// TIA Portal project "BancoProvaProfilometroSpessimetro_V15" (V15)

(* hardware
DEVICE "S71500/ET200MP station_1"  S7-1500 station
   slot 0: "Telaio di montaggio_0"  Rack  6ES7 590-1***0-0AA0
   slot 1: "PLC_1"  CPU 1515-2 PN  6ES7 515-2AM01-0AB0  V2.1
      slot 3: "Display CPU_1"  6ES7591-1BA00-0AA0
DEVICE "GSD device_1"  GSD.Device.PN
   slot 0: "Telaio di montaggio"  Rail  V1.0
   slot 0: "IAI-PRT"  IAI-PRT
   slot 1: "Input 1 word_1"  IAI-PRT
   slot 2: "Input 1 word_2"  IAI-PRT
   slot 3: "Input 1 word_3"  IAI-PRT
   slot 4: "Input 1 word_4"  IAI-PRT
   slot 5: "Input 1 word_5"  IAI-PRT
   slot 6: "Input 1 word_6"  IAI-PRT
   slot 7: "Input 1 word_7"  IAI-PRT
   slot 8: "Input 1 word_8"  IAI-PRT
   slot 9: "Input 1 word_9"  IAI-PRT
   slot 10: "Input 1 word_10"  IAI-PRT
   slot 11: "Input 1 word_11"  IAI-PRT
   slot 12: "Input 1 word_12"  IAI-PRT
   slot 13: "Input 1 word_13"  IAI-PRT
   slot 14: "Input 1 word_14"  IAI-PRT
   slot 15: "Input 1 word_15"  IAI-PRT
   slot 16: "Input 1 word_16"  IAI-PRT
   slot 17: "Output 1 word_1"  IAI-PRT
   slot 18: "Output 1 word_2"  IAI-PRT
   slot 19: "Output 1 word_3"  IAI-PRT
   slot 20: "Output 1 word_4"  IAI-PRT
   slot 21: "Output 1 word_5"  IAI-PRT
   slot 22: "Output 1 word_6"  IAI-PRT
   slot 23: "Output 1 word_7"  IAI-PRT
   slot 24: "Output 1 word_8"  IAI-PRT
   slot 25: "Output 1 word_9"  IAI-PRT
   slot 26: "Output 1 word_10"  IAI-PRT
   slot 27: "Output 1 word_11"  IAI-PRT
   slot 28: "Output 1 word_12"  IAI-PRT
   slot 29: "Output 1 word_13"  IAI-PRT
   slot 30: "Output 1 word_14"  IAI-PRT
   slot 31: "Output 1 word_15"  IAI-PRT
   slot 32: "Output 1 word_16"  IAI-PRT
DEVICE "HMI_1"  KTP400 Comfort
   slot 0: "HMI_1"  KTP400 Comfort  6AV2 124-2DC01-0AX0  15.0.0.0
   slot 1: "HMI_RT_1"  KTP400 Comfort  6AV2 124-2DC01-0AX0  15.0.0.0
   slot 5: "HMI_1.IE_CP_1"  PROFINET Interface  15.0.0.0
      slot 1: "PROFINET Interface_1"  PROFINET Interface
         slot 1: "Porta_1"  Port
   slot 7: "HMI_1.MPI/DP_CP_1"  MPI/DP Interface  15.0.0.0
DEVICE "GSD device_2"  GSD.Device.PN
   slot 0: "Telaio di montaggio"  Rail  V1.0
   slot 0: "dl-pn1"  DL-PN1  1.00
*)

// ===== PLC "PLC_1"  CPU 1515-2 PN =====

VAR_GLOBAL   // PLC tag table "IO_IAI_Controller"
   "RMDS" AT %I30.0 : Bool;   // Stato del segnale operativo - 0: Auto - 1: Manu
   "TRQS" AT %I30.1 : Bool;   // Stato del livello di coppia - questo segnale diventerà vero quando il motore raggiungerà il livello di soglia
   "LOAD" AT %I30.2 : Bool;   // Questo segnale diventerà vero quando la coppia di comando supera la soglia, mentre l'attuatore si trova al interno del range di verifica
   "PZONE" AT %I30.3 : Bool;   // Questo segnale diventerà vero quando dopo l'immissione di un comando di position movement , la posizione effettiva sarà nel range specificato. Uscito da tale range il segnale diventerà falso
   "ZONE1" AT %I30.4 : Bool;   // Questo segnale diventerà vero una volta entrati nel range specificato e sempre solo dopo che l'asse si sia mosso dalla zona 0 (Home) fino alla zona desiderata. Uscito da tale range il contatto diventa falso
   "ZONE2" AT %I30.5 : Bool;   // Questo segnale diventerà vero una volta entrati nel range specificato e sempre solo dopo che l'asse si sia mosso dalla zona 0 (Home) fino alla zona desiderata. Uscito da tale range il contatto diventa falso
   "PWRT" AT %I30.6 : Bool;   // Scrittura della posizione corrente - Se il segnale rimane vero per più di 20ms la posizione attuale verrà salvata da pc1 a pc32
   "EMGS" AT %I30.7 : Bool;   // Stop di emergenza, se viene premuto questa entrata diventa vera
   "PEND" AT %I31.0 : Bool;   // Diventa vero quando il posizionamento è stato terminato
   "HEND" AT %I31.1 : Bool;   // Diventa vero quando viene premuto HOME e l'attuatore è effettivamente nella posizione HOME
   "MOVE" AT %I31.2 : Bool;   // Determina il movimento generico del asse
   "ALM" AT %I31.3 : Bool;   // Contatto NC - se è presente un evento di allarme il segnale diventa falso, in condizioni normali è vero
   "SV" AT %I31.4 : Bool;   // Se vero, indica che il controller è pronto
   "PSFL" AT %I31.5 : Bool;   // -
   "PUSH" AT %I31.6 : Bool;   // -
   "GHMS" AT %I31.7 : Bool;   // -
   "COMMAND_CURRENT" AT %ID4 : DWord;   // Comando attuale
   "CURRENT_SPEED" AT %ID8 : DWord;   // Velocità attuale
   "CSTR" AT %Q31.0 : Bool;   // Start del comando
   "HOME" AT %Q31.1 : Bool;   // L'operazione di ritorno viene avviata a un fronte di salita di questo segnale
   "STP" AT %Q31.2 : Bool;   // ON: l'attuatore può essere spostato, OFF: l'attuatore decelera fino all'arresto
   "RES" AT %Q31.3 : Bool;   // Un allarme viene resettato su un fronte di salita di questo segnale
   "SON" AT %Q31.4 : Bool;   // Servo ON - abilita il servo motore
   "JISL" AT %Q31.5 : Bool;   // Abilita le operazioni manuali (Controller su MANUAL)
   "JVEL" AT %Q31.6 : Bool;
   "JOGneg" AT %Q31.7 : Bool;   // Muovo in libertà l'asse, verso negativo
   "JOGpos" AT %Q30.0 : Bool;   // Muovo in libertà l'asse, verso positivo
   "RMDO" AT %Q30.6 : Bool;   // Questo segnale cambia la modalità operativa tra AUTO e MANU
   "BKRL" AT %Q30.7 : Bool;   // Questo segnale viene utilizzato su un attuatore dotato di un freno per forzarne il rilascio
   "TARGET_POSITION" AT %QD0 : DInt;   // Posizione desiderata
   "POSITION_BAND" AT %QD4 : DInt;   // Banda di posizione desiderata
   "SPEED" AT %QD8 : DInt;   // Veocità simulata
   "ZONE_OUTPUT_POS_positive" AT %QD12 : DInt;
   "ZONE_OUTPUT_POS_negative" AT %QD16 : DInt;
   "PRESSING_CURRENT_LIMIT" AT %QD32 : DInt;
   "LOAD_CURRENT_THRESHOLD" AT %QD36 : DInt;
   "Tag_7" AT %QD26 : DWord;
   "Tag_8" AT %QW24 : Word;
   "ACELERATION" AT %QW20 : Int;   // Accelerzione simulata
   "DECELERATION" AT %QW22 : Int;   // Decelerazione simulata
   "M_SON_AXIS" AT %M100.0 : Bool;
   "M_STR_AXIS" AT %M100.1 : Bool;
   "M_DSTR_ON" AT %M100.2 : Bool;
   "Tag_4" AT %MW32 : Word;
   "Tag_6" AT %MW202 : Word;
   "Tag_12" AT %M204.3 : Bool;
   "Tag_13" AT %MW206 : Word;
   "M_REQUEST_STATUS" AT %M300.0 : Bool;
   "M_RETURN_HOME" AT %M400.0 : Bool;
   "M_JOG_POS" AT %M100.3 : Bool;
   "M_JOG_NEG" AT %M100.4 : Bool;
   "M_RESET_ALLARM" AT %M100.5 : Bool;
   "ON" AT %M106.0 : Bool;
   "Clock_Byte" AT %MB0 : Byte;
   "Clock_10Hz" AT %M0.0 : Bool;
   "Clock_5Hz" AT %M0.1 : Bool;
   "Clock_2.5Hz" AT %M0.2 : Bool;
   "Clock_2Hz" AT %M0.3 : Bool;
   "Clock_1.25Hz" AT %M0.4 : Bool;
   "Clock_1Hz" AT %M0.5 : Bool;
   "Clock_0.625Hz" AT %M0.6 : Bool;
   "Clock_0.5Hz" AT %M0.7 : Bool;
   "Tag_1" AT %M120.0 : Bool;
   "System_Byte" AT %MB1 : Byte;
   "FirstScan" AT %M1.0 : Bool;
   "DiagStatusUpdate" AT %M1.1 : Bool;
   "AlwaysTRUE" AT %M1.2 : Bool;
   "AlwaysFALSE" AT %M1.3 : Bool;
   "ReportFF" AT %M410.0 : Bool;
   "SelectOPMode" AT %M10.0 : Bool;   // Seleziono il modo operativo
   "OPMode_Set" AT %M10.1 : Bool;   // Porto a 1 il modo operativo
   "OPMode_Reset" AT %M10.2 : Bool;   // Porto a 0 il modo operativo
   "OPMode_ResetCTU" AT %M10.3 : Bool;   // Resetto il conteggio di Counter_JogAuto
   "Rnd_Seed" AT %MW100 : Word;
   "Rnd_Restart" AT %M20.0 : Bool;
   "Rnd_Record" AT %MW101 : Word;
   "Rnd_Seed_Pos" AT %MW102 : Word;
   "Rnd_Record_Pos" AT %MW113 : Word;
   "Restart_Sim" AT %M30.0 : Bool;
   "Restart_Sim_Set" AT %M30.1 : Bool;
   "Restart_Sim_Reset" AT %M30.2 : Bool;
   "Restart_Sim_RCTU" AT %M30.3 : Bool;
   "PreviusPosition" AT %MD103 : DWord;
   "ChangeDetected" AT %M40.0 : Bool;
   "Tag_5" AT %MD104 : DWord;
   "ResetSQLChangeValue" AT %M50.0 : Bool;
   "REQ_IL1000_Set" AT %M60.0 : Bool;
   "REQ_IL1000_Reset" AT %M60.1 : Bool;
   "REQ_IL1000_ResCTU" AT %M60.2 : Bool;
   "Tag_2" AT %M70.0 : Bool;
   "Tag_3" AT %M80.0 : Bool;
   "Tag_9" AT %MD45 : DWord;
   "Tag_10" AT %MD46 : DWord;
   "Tag_11" AT %M5.0 : Bool;
   "Simu_Timer" AT %M6.0 : Bool;
   "RawPosition" AT %ID0 : DWord;
   "M_SON" AT %M101.0 : Bool;   // Merker - Start Servo
   "Cock_10Hz_Neg" AT %M321.0 : Bool;
   "Tag_16" AT %M102.0 : Bool;
END_VAR

VAR_GLOBAL   // PLC tag table "Keyence"
   "SensorIN" AT %IW32 : Word;
   "ERROR_IL1000" AT %M204.2 : Bool;
   "RECORD_IL1000" AT %MD215 : DInt;
   "LEN_IL1000" AT %MD210 : DWord;
   "STATUS_IL1000" AT %MD206 : DWord;
   "VALID_IL1000" AT %M204.0 : Bool;
   "BUSY_IL1000" AT %M204.1 : Bool;
   "REQ_IL1000" AT %M500.0 : Bool;
   "IL_100_ST" AT %M100.6 : Bool;
END_VAR

// folder: Database/Istanze

DATA_BLOCK "Output_DB"   // DB7
{ S7_Optimized_Access := 'TRUE' }
AUTHOR : Valentino-Fabbri
VERSION : 0.1
// stored: InstanceOfName Output
"Output"
BEGIN
END_DATA_BLOCK

DATA_BLOCK "Jog Manager_DB"   // DB8
{ S7_Optimized_Access := 'TRUE' }
AUTHOR : Valentino-Fabbri
VERSION : 0.1
// stored: InstanceOfName Jog Manager
"Jog Manager"
BEGIN
END_DATA_BLOCK

DATA_BLOCK "Position Move_DB"   // DB9
{ S7_Optimized_Access := 'TRUE' }
AUTHOR : Valentino-Fabbri
VERSION : 0.1
// stored: InstanceOfName Position Move
"Position Move"
BEGIN
END_DATA_BLOCK

DATA_BLOCK "Speed Move_DB"   // DB10
{ S7_Optimized_Access := 'TRUE' }
AUTHOR : Valentino-Fabbri
VERSION : 0.1
// stored: InstanceOfName Speed Move
"Speed Move"
BEGIN
END_DATA_BLOCK

DATA_BLOCK "DoubleTapButton2_DB_3"   // DB12
{ S7_Optimized_Access := 'TRUE' }
VERSION : 0.1
// stored: InstanceOfName DoubleTapButton2
"DoubleTapButton2"
BEGIN
END_DATA_BLOCK

DATA_BLOCK "DoubleTapButton2_DB"   // DB21
{ S7_Optimized_Access := 'TRUE' }
VERSION : 0.1
// stored: InstanceOfName DoubleTapButton2
"DoubleTapButton2"
BEGIN
END_DATA_BLOCK

DATA_BLOCK "DoubleTapButton2_DB_1"   // DB22
{ S7_Optimized_Access := 'TRUE' }
VERSION : 0.1
// stored: InstanceOfName DoubleTapButton2
"DoubleTapButton2"
BEGIN
END_DATA_BLOCK

DATA_BLOCK "DoubleTapButton2_DB_2"   // DB23
{ S7_Optimized_Access := 'TRUE' }
VERSION : 0.1
// stored: InstanceOfName DoubleTapButton2
"DoubleTapButton2"
BEGIN
END_DATA_BLOCK

DATA_BLOCK "CollisionMovement_DB"   // DB24
{ S7_Optimized_Access := 'TRUE' }
AUTHOR : Valentino-Fabbri
VERSION : 0.1
// stored: InstanceOfName CollisionMovement
"CollisionMovement"
BEGIN
END_DATA_BLOCK

DATA_BLOCK "Input_DB"   // DB26
{ S7_Optimized_Access := 'TRUE' }
AUTHOR : Valentino-Fabbri
VERSION : 0.1
// stored: InstanceOfName Input
"Input"
BEGIN
END_DATA_BLOCK

// folder: Database/Static

DATA_BLOCK "IAI_DATI"   // DB2
{ S7_Optimized_Access := 'TRUE' }
VERSION : 0.1
   VAR
      "TargetPosition 1" : DInt := 0;   // Posizione desiderata - impostata a metà
      "TargetPosition 2" : Real := 0.0;
      "TargetPosition 2 Out" : DInt;
      PositionBand : Real := 10000.0;   // Margine di errore sulla posizione desiderata
      PositionBandOut : DInt;
      Speed : Real := 3000.0;   // Velocità espressa in mm/s
      SpeedOut : DInt := 0;
      Aceleration : Real := 1.0;   // Accellerazione
      AcelerationOut : DInt := 0;
      Deceleration : Real := 1.0;   // Decellerazione
      DecelerationOut : DInt := 0;
      ZonePos : Real := 10000.0;
      ZonePosOut : DInt := 0;
      ZoneNeg : Real := 10000.0;
      ZoneNegOut : DInt;
      Speed_JOG : Real := 15000.0;   // Velocità espressa in mm/s
      Speed_JOG_Out : DInt;
      Aceleration_JOG : Real := 5.0;   // Accellerazione
      Aceleration_JOG_Out : DInt;
      Deceleration_JOG : Real := 5.0;   // Decellerazione
      Deceleration_JOG_Out : DInt;
      ActualPosition : Real;
      ModoOperativo : Bool;   // 0=Auto 1=Jog
      PN_Start : Int;
      WrongPositionBand : Bool;
      WrongTargetPosition2 : Bool;
      WrongZonePos : Bool;
      WrongZoneNeg : Bool;
      WrongSpeed : Bool;
      WrongAceleration : Bool;
      WrongDeceleration : Bool;
      ErrPositionBand : Bool;
      ErrSpeed : Bool;
      ErrDeceleration : Bool;
      ErrAceleration : Bool;
      ErrZonePos : Bool;
      ErrZoneNeg : Bool;
      ErrTargetPosition2 : Bool;
      PositionBandHighLimit : Real := 20030.0;
      PositionBandLowLimit : Real := 5.0;
      SpeedHighLimit : Real := 90000.0;
      SpeedLowLimit : Real := 1.0;
      AcelerationHighLimit : Real := 10.0;
      AcelerationLowLimit : Real := 1.0;
      DecelerationHighLimit : Real := 10.0;
      DecelerationLowLimit : Real := 1.0;
      TargetPosition2HighLimit : Real := 20015.0;
      TargetPosition2LowLimit : Real := -15.0;
      ZonePosHighLimit : Real := 999999.0;
      ZonePosLowLimit : Real := -999999.0;
      ZoneNegHighLimit : Real := 999999.0;
      ZoneNegLowLimit : Real := -999999.0;
      PositionEnd : Bool;
   END_VAR
BEGIN
END_DATA_BLOCK

DATA_BLOCK "Keyence_DATI"   // DB3
{ S7_Optimized_Access := 'TRUE' }
VERSION : 0.1
   VAR
      MeasureValue : Real;
      Request : Bool;
      ARLM_IL_1000 : Int;   // Anomalia generica - lettura amplificatore Keyence
      Record : DInt;
      Id : Hw_Io := 16#12F;
      Index : DInt := 38;
      MLen : DInt := 4;
      IsValid : Bool;
      IsBusy : Bool;
      IsError : Bool;
      Status : DWord;
      Activate : Bool;
      Lenght : DWord;
      EnableLog : Bool;
      ReadError : Bool;
   END_VAR
BEGIN
END_DATA_BLOCK

DATA_BLOCK "Rugosimetro"   // DB4
{ S7_Optimized_Access := 'TRUE' }
VERSION : 0.1
   VAR
      Ra : Real;
      "Counter" : Real;
      Accumulatore : Real;
      Difu1 : Bool;
      Difu2 : Bool;
      ValoreAttualeModulo : Real;
      difu3 : Bool;
   END_VAR
BEGIN
END_DATA_BLOCK

DATA_BLOCK "SQL"   // DB11
TITLE = Sql
{ S7_Optimized_Access := 'TRUE' }
AUTHOR : Valentino-Fabbri
VERSION : 0.1
   VAR
      ChangeValue : Bool;
      SendValue : Time := T#500ms;
      SetName : String[10];
      Simulation : Bool;
      CTUPos : Real;
      CTUAlt : Real;
      SendFile : Int;
      BtnSend : Bool;
      CheckState : Int;
   END_VAR
BEGIN
END_DATA_BLOCK

DATA_BLOCK "Simulation"   // DB20
{ S7_Optimized_Access := 'TRUE' }
VERSION : 0.1
   VAR
      HighMax : DWord := 5;
      PositionMax : DWord := 200;
      SimuTimeIn : Time := T#10s;
      SimuTimeOut : Time;
      SimuTimer : Bool;
   END_VAR
BEGIN
END_DATA_BLOCK

// folder: System blocks/Program resources

DATA_BLOCK "IEC_Timer_0_DB"   // DB5
{ S7_Optimized_Access := 'TRUE' }
AUTHOR : Simatic
FAMILY : IEC
NAME : IEC_TMR
VERSION : 1.0
// stored: InstanceOfName IEC_TIMER
"IEC_TIMER"
BEGIN
END_DATA_BLOCK

DATA_BLOCK "IEC_Timer_0_DB_1"   // DB6
{ S7_Optimized_Access := 'TRUE' }
AUTHOR : Simatic
FAMILY : IEC
NAME : IEC_TMR
VERSION : 1.0
// stored: InstanceOfName IEC_TIMER
"IEC_TIMER"
BEGIN
END_DATA_BLOCK

DATA_BLOCK "IEC_Counter_0_DB"   // DB13
{ S7_Optimized_Access := 'TRUE' }
AUTHOR : Simatic
FAMILY : IEC
NAME : CNTR
VERSION : 1.0
// stored: InstanceOfName IEC_COUNTER
"IEC_COUNTER"
BEGIN
END_DATA_BLOCK

DATA_BLOCK "Counter_EnableRequest"   // DB14
{ S7_Optimized_Access := 'TRUE' }
AUTHOR : Simatic
FAMILY : IEC
NAME : CNTR
VERSION : 1.0
// stored: InstanceOfName IEC_COUNTER
"IEC_COUNTER"
BEGIN
END_DATA_BLOCK

DATA_BLOCK "IEC_Timer_0_DB_2"   // DB15
{ S7_Optimized_Access := 'TRUE' }
AUTHOR : Simatic
FAMILY : IEC
NAME : IEC_TMR
VERSION : 1.0
// stored: InstanceOfName IEC_TIMER
"IEC_TIMER"
BEGIN
END_DATA_BLOCK

DATA_BLOCK "IEC_Timer_0_DB_3"   // DB16
{ S7_Optimized_Access := 'TRUE' }
AUTHOR : Simatic
FAMILY : IEC
NAME : IEC_TMR
VERSION : 1.0
// stored: InstanceOfName IEC_TIMER
"IEC_TIMER"
BEGIN
END_DATA_BLOCK

DATA_BLOCK "IEC_Counter_0_DB_1"   // DB17
{ S7_Optimized_Access := 'TRUE' }
AUTHOR : Simatic
FAMILY : IEC
NAME : CNTR
VERSION : 1.0
// stored: InstanceOfName IEC_COUNTER
"IEC_COUNTER"
BEGIN
END_DATA_BLOCK

DATA_BLOCK "IEC_Counter_0_DB_2"   // DB18
{ S7_Optimized_Access := 'TRUE' }
AUTHOR : Simatic
FAMILY : IEC
NAME : CNTR
VERSION : 1.0
// stored: InstanceOfName IEC_COUNTER
"IEC_COUNTER"
BEGIN
END_DATA_BLOCK

DATA_BLOCK "IEC_Timer_0_DB_4"   // DB19
{ S7_Optimized_Access := 'TRUE' }
AUTHOR : Simatic
FAMILY : IEC
NAME : IEC_TMR
VERSION : 1.0
// stored: InstanceOfName IEC_TIMER
"IEC_TIMER"
BEGIN
END_DATA_BLOCK

DATA_BLOCK "IEC_Timer_0_DB_5"   // DB25
{ S7_Optimized_Access := 'TRUE' }
AUTHOR : Simatic
FAMILY : IEC
NAME : IEC_TMR
VERSION : 1.0
// stored: InstanceOfName IEC_TIMER
"IEC_TIMER"
BEGIN
END_DATA_BLOCK

// folder: (top level)

ORGANIZATION_BLOCK "Main"   // OB1, LAD, ProgramCycle
TITLE = "Main Program Sweep (Cycle)"
{ S7_Optimized_Access := 'TRUE' }
VERSION : 0.1
   VAR_INPUT
      Initial_Call : Bool;   // Initial call of this OB
      Remanence : Bool;   // =True, if remanent data are available
   END_VAR
   VAR_TEMP   // added for the SCL form of the ladder/FBD networks
      _w1 : Bool;
   END_VAR
BEGIN

REGION Network 1: Assegno gli Output
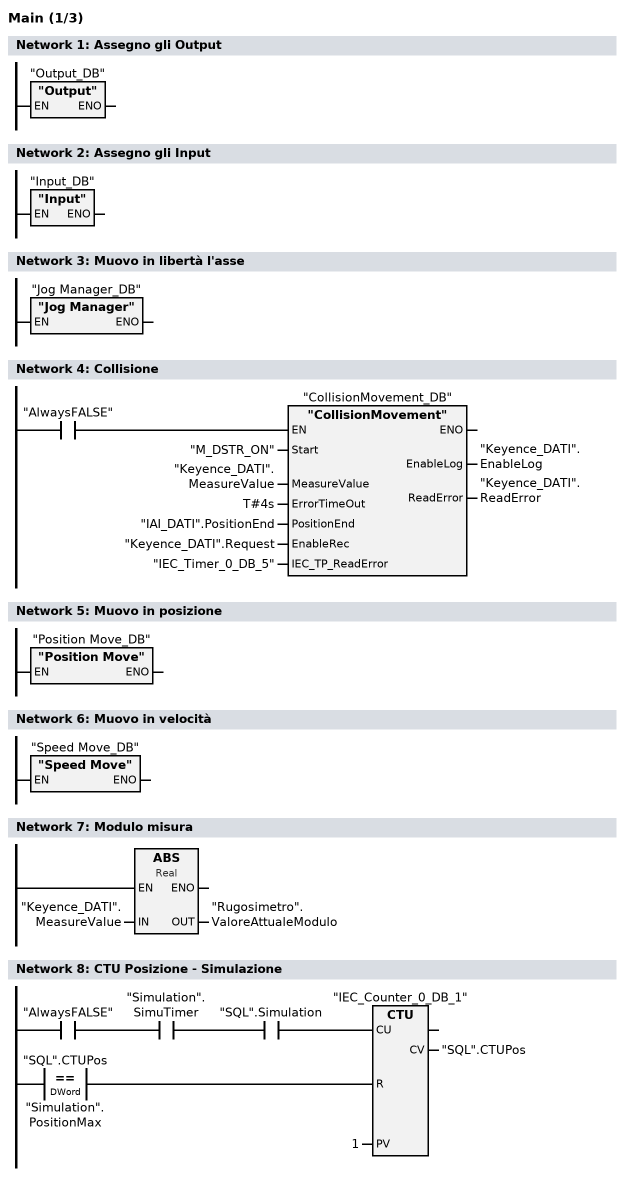
   RUNG wire#powerrail
      "Output_DB"()
   END_RUNG
   // the same network as SCL:
   "Output_DB"();   // "Output"
END_REGION

REGION Network 2: Assegno gli Input
   RUNG wire#powerrail
      "Input_DB"()
   END_RUNG
   // the same network as SCL:
   "Input_DB"();   // "Input"
END_REGION

REGION Network 3: Muovo in libertà l'asse
   RUNG wire#powerrail
      "Jog Manager_DB"()
   END_RUNG
   // the same network as SCL:
   "Jog Manager_DB"();   // "Jog Manager"
END_REGION

REGION Network 4: Collisione
   RUNG wire#powerrail
      Contact( "AlwaysFALSE" )
      "CollisionMovement_DB"(Start := "M_DSTR_ON", MeasureValue := "Keyence_DATI".MeasureValue, ErrorTimeOut := T#4s, PositionEnd := "IAI_DATI".PositionEnd, EnableRec := "Keyence_DATI".Request, IEC_TP_ReadError := "IEC_Timer_0_DB_5", EnableLog => "Keyence_DATI".EnableLog, ReadError => "Keyence_DATI".ReadError)
   END_RUNG
   // the same network as SCL:
   IF "AlwaysFALSE" THEN
       "CollisionMovement_DB"(Start := "M_DSTR_ON",   // "CollisionMovement"
                              MeasureValue := "Keyence_DATI".MeasureValue,
                              ErrorTimeOut := T#4s,
                              PositionEnd := "IAI_DATI".PositionEnd,
                              EnableRec := "Keyence_DATI".Request,
                              IEC_TP_ReadError := "IEC_Timer_0_DB_5",
                              EnableLog => "Keyence_DATI".EnableLog,
                              ReadError => "Keyence_DATI".ReadError);
   END_IF;
END_REGION

REGION Network 5: Muovo in posizione
   RUNG wire#powerrail
      "Position Move_DB"()
   END_RUNG
   // the same network as SCL:
   "Position Move_DB"();   // "Position Move"
END_REGION

REGION Network 6: Muovo in velocità
   RUNG wire#powerrail
      "Speed Move_DB"()
   END_RUNG
   // the same network as SCL:
   "Speed Move_DB"();   // "Speed Move"
END_REGION

REGION Network 7: Modulo misura
   RUNG wire#powerrail
      { S7_Templates := "SrcType := Real" } Abs(in := "Keyence_DATI".MeasureValue, out => "Rugosimetro".ValoreAttualeModulo)
   END_RUNG
   // the same network as SCL:
   "Rugosimetro".ValoreAttualeModulo := ABS("Keyence_DATI".MeasureValue);
END_REGION

REGION Network 8: CTU Posizione - Simulazione
   "IEC_Counter_0_DB_1".CTU(CU := "AlwaysFALSE" AND "Simulation".SimuTimer AND "SQL".Simulation,
                           R := "SQL".CTUPos = "Simulation".PositionMax,
                           PV := 1,
                           CV => "SQL".CTUPos);
END_REGION

REGION Network 9: CTU Altezza - Simulazione
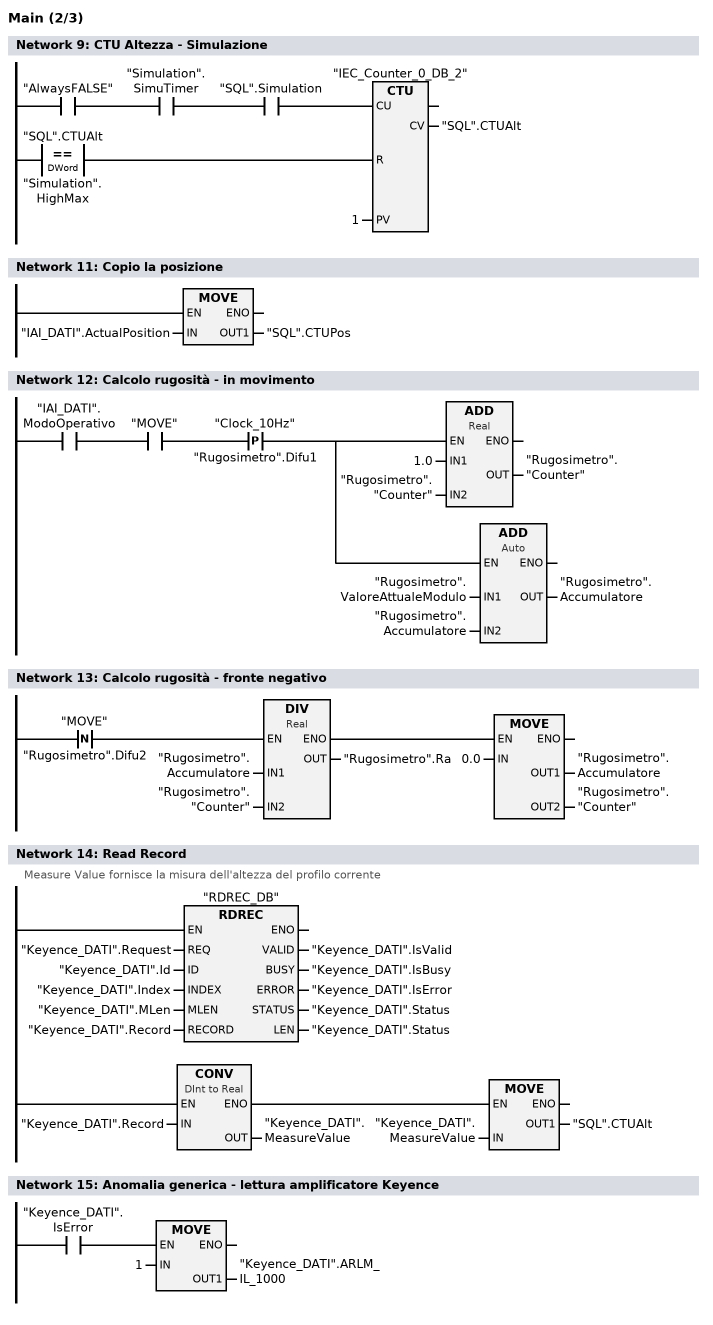
   "IEC_Counter_0_DB_2".CTU(CU := "AlwaysFALSE" AND "Simulation".SimuTimer AND "SQL".Simulation,
                           R := "SQL".CTUAlt = "Simulation".HighMax,
                           PV := 1,
                           CV => "SQL".CTUAlt);
END_REGION

REGION Network 10 (STL): Scalo la posizione
   // %ID0 - Simulazione: %MD3000
   // ActualPosition fornisce una misura della posizione corrente
         L     "RawPosition";
         DTR;
         L     100.0;
         /R;
         T     "IAI_DATI".ActualPosition;
END_REGION

REGION Network 11: Copio la posizione
   RUNG wire#powerrail
      Move(in := "IAI_DATI".ActualPosition, out1 => "SQL".CTUPos)
   END_RUNG
   // the same network as SCL:
   "SQL".CTUPos := "IAI_DATI".ActualPosition;
END_REGION

REGION Network 12: Calcolo rugosità - in movimento
   RUNG wire#powerrail
      Contact( "IAI_DATI".ModoOperativo )
      Contact( "MOVE" )
      P_Contact(operand := "Clock_10Hz", bit := "Rugosimetro".Difu1)
      wire#w1
      { S7_Templates := "SrcType := Real" } Add(in1 := 1.0, in2 := "Rugosimetro"."Counter", out => "Rugosimetro"."Counter")
   END_RUNG
   RUNG wire#w1
      Add(in1 := "Rugosimetro".ValoreAttualeModulo, in2 := "Rugosimetro".Accumulatore, out => "Rugosimetro".Accumulatore)
   END_RUNG
   // the same network as SCL:
   #_w1 := "IAI_DATI".ModoOperativo AND "MOVE" AND "Clock_10Hz" AND NOT "Rugosimetro".Difu1;   // rising edge of "Clock_10Hz"
   "Rugosimetro".Difu1 := "Clock_10Hz";
   IF #_w1 THEN
       "Rugosimetro"."Counter" := 1.0 + "Rugosimetro"."Counter";
       "Rugosimetro".Accumulatore := "Rugosimetro".ValoreAttualeModulo + "Rugosimetro".Accumulatore;
   END_IF;
END_REGION

REGION Network 13: Calcolo rugosità - fronte negativo
   RUNG wire#powerrail
      N_Contact(operand := "MOVE", bit := "Rugosimetro".Difu2)
      { S7_Templates := "SrcType := Real" } Div(in1 := "Rugosimetro".Accumulatore, in2 := "Rugosimetro"."Counter", out => "Rugosimetro".Ra)
      Move(in := 0.0, out1 => "Rugosimetro".Accumulatore, out2 => "Rugosimetro"."Counter")
   END_RUNG
   // the same network as SCL:
   #_w1 := NOT "MOVE" AND "Rugosimetro".Difu2;   // falling edge of "MOVE"
   "Rugosimetro".Difu2 := "MOVE";
   IF #_w1 THEN
       "Rugosimetro".Ra := "Rugosimetro".Accumulatore / "Rugosimetro"."Counter";
       "Rugosimetro".Accumulatore := 0.0;
       "Rugosimetro"."Counter" := 0.0;
   END_IF;
END_REGION

REGION Network 14: Read Record
   // Measure Value fornisce la misura dell'altezza del profilo corrente
   "RDREC_DB"(REQ := "Keyence_DATI".Request,   // RDREC
              ID := "Keyence_DATI".Id,
              INDEX := "Keyence_DATI".Index,
              MLEN := "Keyence_DATI".MLen,
              RECORD := "Keyence_DATI".Record,
              VALID => "Keyence_DATI".IsValid,
              BUSY => "Keyence_DATI".IsBusy,
              ERROR => "Keyence_DATI".IsError,
              STATUS => "Keyence_DATI".Status,
              LEN => "Keyence_DATI".Status);
   "Keyence_DATI".MeasureValue := DINT_TO_REAL("Keyence_DATI".Record);
   "SQL".CTUAlt := "Keyence_DATI".MeasureValue;
END_REGION

REGION Network 15: Anomalia generica - lettura amplificatore Keyence
   RUNG wire#powerrail
      Contact( "Keyence_DATI".IsError )
      Move(in := 1, out1 => "Keyence_DATI".ARLM_IL_1000)
   END_RUNG
   // the same network as SCL:
   IF "Keyence_DATI".IsError THEN "Keyence_DATI".ARLM_IL_1000 := 1; END_IF;
END_REGION

REGION Network 16: Resetto l'anomalia
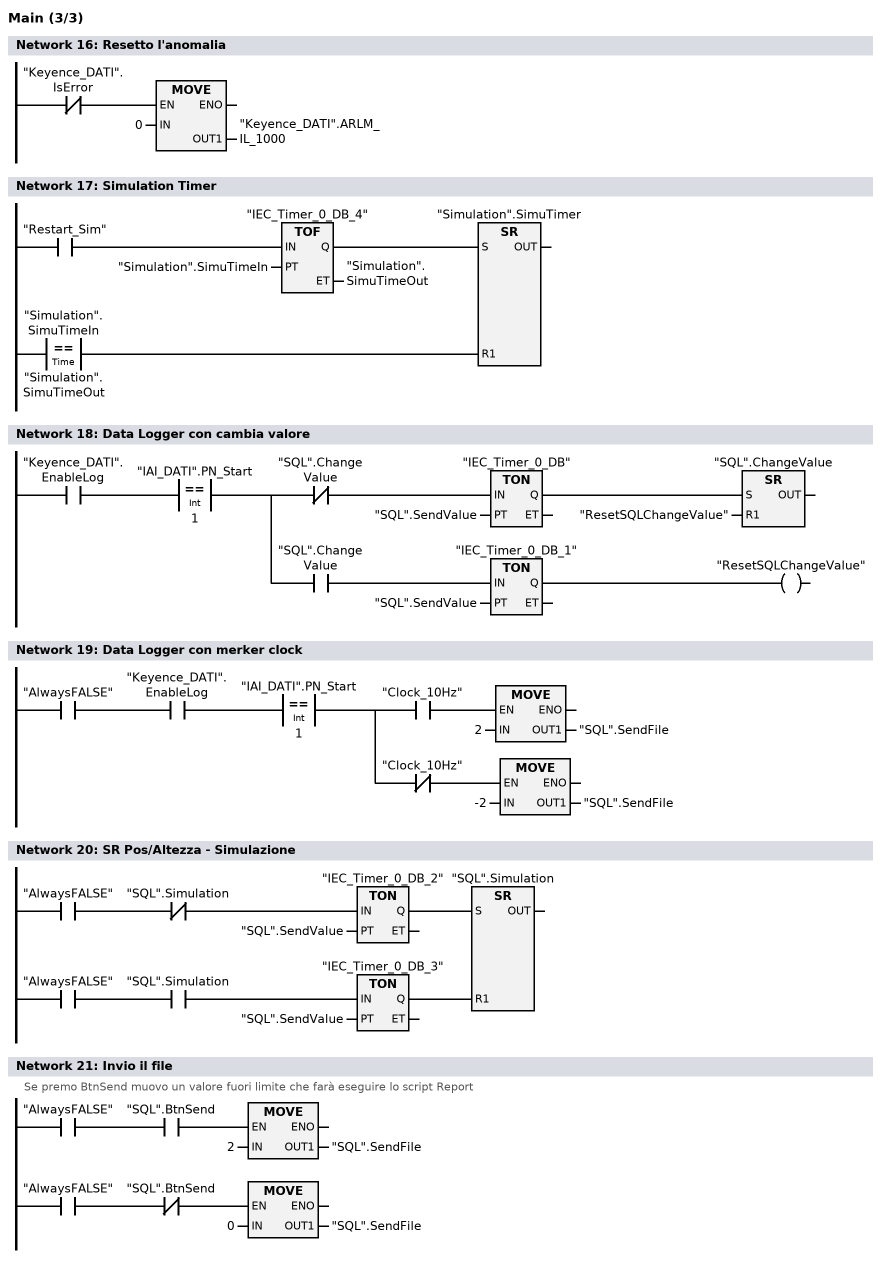
   RUNG wire#powerrail
      I_Contact( "Keyence_DATI".IsError )
      Move(in := 0, out1 => "Keyence_DATI".ARLM_IL_1000)
   END_RUNG
   // the same network as SCL:
   IF NOT "Keyence_DATI".IsError THEN "Keyence_DATI".ARLM_IL_1000 := 0; END_IF;
END_REGION

REGION Network 17: Simulation Timer
   "IEC_Timer_0_DB_4".TOF(IN := "Restart_Sim", PT := "Simulation".SimuTimeIn, ET => "Simulation".SimuTimeOut);
   IF "IEC_Timer_0_DB_4".Q THEN
       "Simulation".SimuTimer := TRUE;   // SR flip-flop
   END_IF;
   IF "Simulation".SimuTimeIn = "Simulation".SimuTimeOut THEN "Simulation".SimuTimer := FALSE; END_IF;
END_REGION

REGION Network 18: Data Logger con cambia valore
   #_w1 := "Keyence_DATI".EnableLog AND ("IAI_DATI".PN_Start = 1);
   "IEC_Timer_0_DB".TON(IN := #_w1 AND NOT "SQL".ChangeValue, PT := "SQL".SendValue);
   IF "IEC_Timer_0_DB".Q THEN
       "SQL".ChangeValue := TRUE;   // SR flip-flop
   END_IF;
   IF "ResetSQLChangeValue" THEN "SQL".ChangeValue := FALSE; END_IF;
   "IEC_Timer_0_DB_1".TON(IN := #_w1 AND "SQL".ChangeValue, PT := "SQL".SendValue);
   "ResetSQLChangeValue" := "IEC_Timer_0_DB_1".Q;
END_REGION

REGION Network 19: Data Logger con merker clock
   RUNG wire#powerrail
      Contact( "AlwaysFALSE" )
      Contact( "Keyence_DATI".EnableLog )
      { S7_Templates := "SrcType := Int" } EQ_Contact(in1 := "IAI_DATI".PN_Start, in2 := 1)
      wire#w1
      Contact( "Clock_10Hz" )
      Move(in := 2, out1 => "SQL".SendFile)
   END_RUNG
   RUNG wire#w1
      I_Contact( "Clock_10Hz" )
      Move(in := -2, out1 => "SQL".SendFile)
   END_RUNG
   // the same network as SCL:
   #_w1 := "AlwaysFALSE" AND "Keyence_DATI".EnableLog AND ("IAI_DATI".PN_Start = 1);
   IF #_w1 AND "Clock_10Hz" THEN "SQL".SendFile := 2; END_IF;
   IF #_w1 AND NOT "Clock_10Hz" THEN "SQL".SendFile := -2; END_IF;
END_REGION

REGION Network 20: SR Pos/Altezza - Simulazione
   "IEC_Timer_0_DB_2".TON(IN := "AlwaysFALSE" AND NOT "SQL".Simulation, PT := "SQL".SendValue);
   "IEC_Timer_0_DB_3".TON(IN := "AlwaysFALSE" AND "SQL".Simulation, PT := "SQL".SendValue);
   IF "IEC_Timer_0_DB_2".Q THEN
       "SQL".Simulation := TRUE;   // SR flip-flop
   END_IF;
   IF "IEC_Timer_0_DB_3".Q THEN "SQL".Simulation := FALSE; END_IF;
END_REGION

REGION Network 21: Invio il file
   // Se premo BtnSend muovo un valore fuori limite che farà eseguire lo script Report
   RUNG wire#powerrail
      Contact( "AlwaysFALSE" )
      Contact( "SQL".BtnSend )
      Move(in := 2, out1 => "SQL".SendFile)
   END_RUNG
   RUNG wire#powerrail
      Contact( "AlwaysFALSE" )
      I_Contact( "SQL".BtnSend )
      Move(in := 0, out1 => "SQL".SendFile)
   END_RUNG
   // the same network as SCL:
   IF "AlwaysFALSE" AND "SQL".BtnSend THEN "SQL".SendFile := 2; END_IF;
   IF "AlwaysFALSE" AND NOT "SQL".BtnSend THEN "SQL".SendFile := 0; END_IF;
END_REGION
END_ORGANIZATION_BLOCK

// folder: Funzionali

FUNCTION_BLOCK "Output"   // FB1, LAD
TITLE = Output
{ S7_Optimized_Access := 'TRUE' }
AUTHOR : Valentino-Fabbri
VERSION : 0.1
   VAR_TEMP   // added for the SCL form of the ladder/FBD networks
      _w1 : Bool;
   END_VAR
BEGIN

REGION Network 1: Servo motore sempre acceso
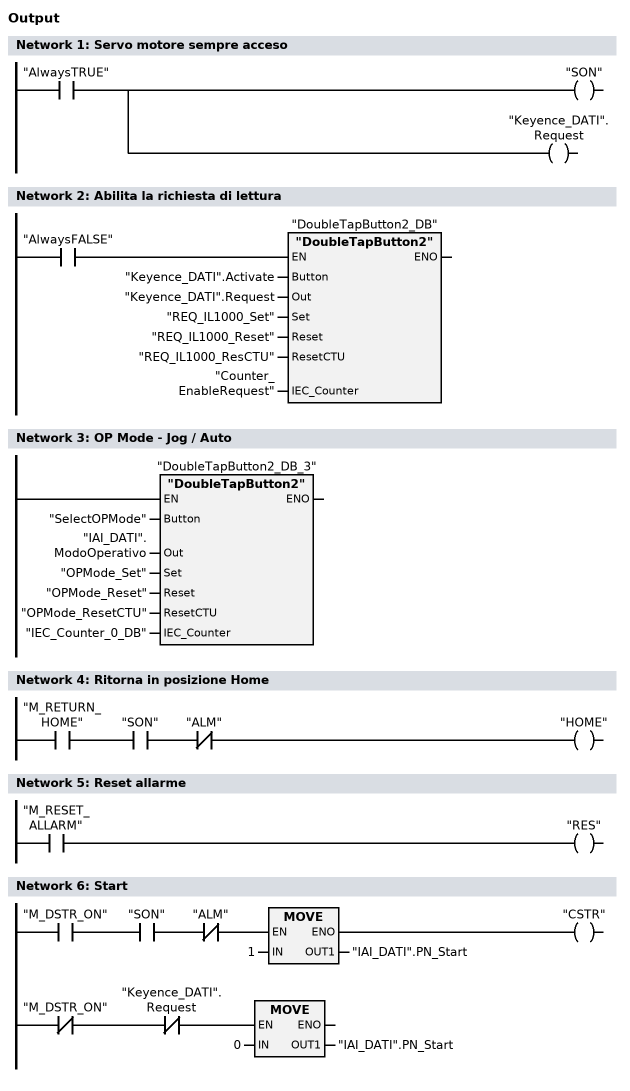
   RUNG wire#powerrail
      Contact( "AlwaysTRUE" )
      wire#w1
      Coil( "SON" )
   END_RUNG
   RUNG wire#w1
      Coil( "Keyence_DATI".Request )
   END_RUNG
   // the same network as SCL:
   "SON" := "AlwaysTRUE";
   "Keyence_DATI".Request := "AlwaysTRUE";
END_REGION

REGION Network 2: Abilita la richiesta di lettura
   RUNG wire#powerrail
      Contact( "AlwaysFALSE" )
      "DoubleTapButton2_DB"(Button := "Keyence_DATI".Activate, Out := "Keyence_DATI".Request, Set := "REQ_IL1000_Set", Reset := "REQ_IL1000_Reset", ResetCTU := "REQ_IL1000_ResCTU", IEC_Counter := "Counter_EnableRequest")
   END_RUNG
   // the same network as SCL:
   IF "AlwaysFALSE" THEN
       "DoubleTapButton2_DB"(Button := "Keyence_DATI".Activate,   // "DoubleTapButton2"
                             Out := "Keyence_DATI".Request,
                             Set := "REQ_IL1000_Set",
                             Reset := "REQ_IL1000_Reset",
                             ResetCTU := "REQ_IL1000_ResCTU",
                             IEC_Counter := "Counter_EnableRequest");
   END_IF;
END_REGION

REGION Network 3: OP Mode - Jog / Auto
   RUNG wire#powerrail
      "DoubleTapButton2_DB_3"(Button := "SelectOPMode", Out := "IAI_DATI".ModoOperativo, Set := "OPMode_Set", Reset := "OPMode_Reset", ResetCTU := "OPMode_ResetCTU", IEC_Counter := "IEC_Counter_0_DB")
   END_RUNG
   // the same network as SCL:
   "DoubleTapButton2_DB_3"(Button := "SelectOPMode",   // "DoubleTapButton2"
                           Out := "IAI_DATI".ModoOperativo,
                           Set := "OPMode_Set",
                           Reset := "OPMode_Reset",
                           ResetCTU := "OPMode_ResetCTU",
                           IEC_Counter := "IEC_Counter_0_DB");
END_REGION

REGION Network 4: Ritorna in posizione Home
   RUNG wire#powerrail
      Contact( "M_RETURN_HOME" )
      Contact( "SON" )
      I_Contact( "ALM" )
      Coil( "HOME" )
   END_RUNG
   // the same network as SCL:
   "HOME" := "M_RETURN_HOME" AND "SON" AND NOT "ALM";
END_REGION

REGION Network 5: Reset allarme
   RUNG wire#powerrail
      Contact( "M_RESET_ALLARM" )
      Coil( "RES" )
   END_RUNG
   // the same network as SCL:
   "RES" := "M_RESET_ALLARM";
END_REGION

REGION Network 6: Start
   RUNG wire#powerrail
      Contact( "M_DSTR_ON" )
      Contact( "SON" )
      I_Contact( "ALM" )
      Move(in := 1, out1 => "IAI_DATI".PN_Start)
      Coil( "CSTR" )
   END_RUNG
   RUNG wire#powerrail
      I_Contact( "M_DSTR_ON" )
      I_Contact( "Keyence_DATI".Request )
      Move(in := 0, out1 => "IAI_DATI".PN_Start)
   END_RUNG
   // the same network as SCL:
   #_w1 := "M_DSTR_ON" AND "SON" AND NOT "ALM";
   IF #_w1 THEN "IAI_DATI".PN_Start := 1; END_IF;
   "CSTR" := #_w1;
   IF NOT "M_DSTR_ON" AND NOT "Keyence_DATI".Request THEN "IAI_DATI".PN_Start := 0; END_IF;
END_REGION
END_FUNCTION_BLOCK

FUNCTION_BLOCK "Jog Manager"   // FB2, LAD
TITLE = Jog Manager
{ S7_Optimized_Access := 'TRUE' }
AUTHOR : Valentino-Fabbri
VERSION : 0.1
   VAR_TEMP   // added for the SCL form of the ladder/FBD networks
      _w1 : Bool;
   END_VAR
BEGIN

REGION Network 1: Muovo in libertà l'asse, verso positivo - verso negativo
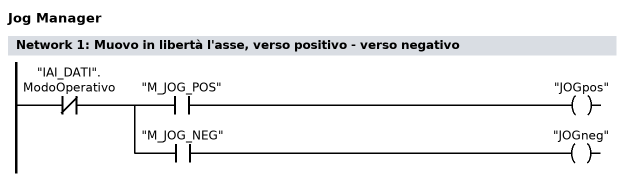
   RUNG wire#powerrail
      I_Contact( "IAI_DATI".ModoOperativo )
      wire#w1
      Contact( "M_JOG_POS" )
      Coil( "JOGpos" )
   END_RUNG
   RUNG wire#w1
      Contact( "M_JOG_NEG" )
      Coil( "JOGneg" )
   END_RUNG
   // the same network as SCL:
   #_w1 := NOT "IAI_DATI".ModoOperativo;
   "JOGpos" := #_w1 AND "M_JOG_POS";
   "JOGneg" := #_w1 AND "M_JOG_NEG";
END_REGION
END_FUNCTION_BLOCK

FUNCTION_BLOCK "Position Move"   // FB3, LAD
TITLE = Position Move
{ S7_Optimized_Access := 'TRUE' }
AUTHOR : Valentino-Fabbri
VERSION : 0.1
   VAR_TEMP   // added for the SCL form of the ladder/FBD networks
      _w1 : Bool;
      _w2 : Bool;
      _w3 : Bool;
      _w4 : Bool;
   END_VAR
BEGIN

REGION Network 1: Simulazione data una posizione
   // Es: Output: %MD0 corrisponde alla double %QD0 e così via
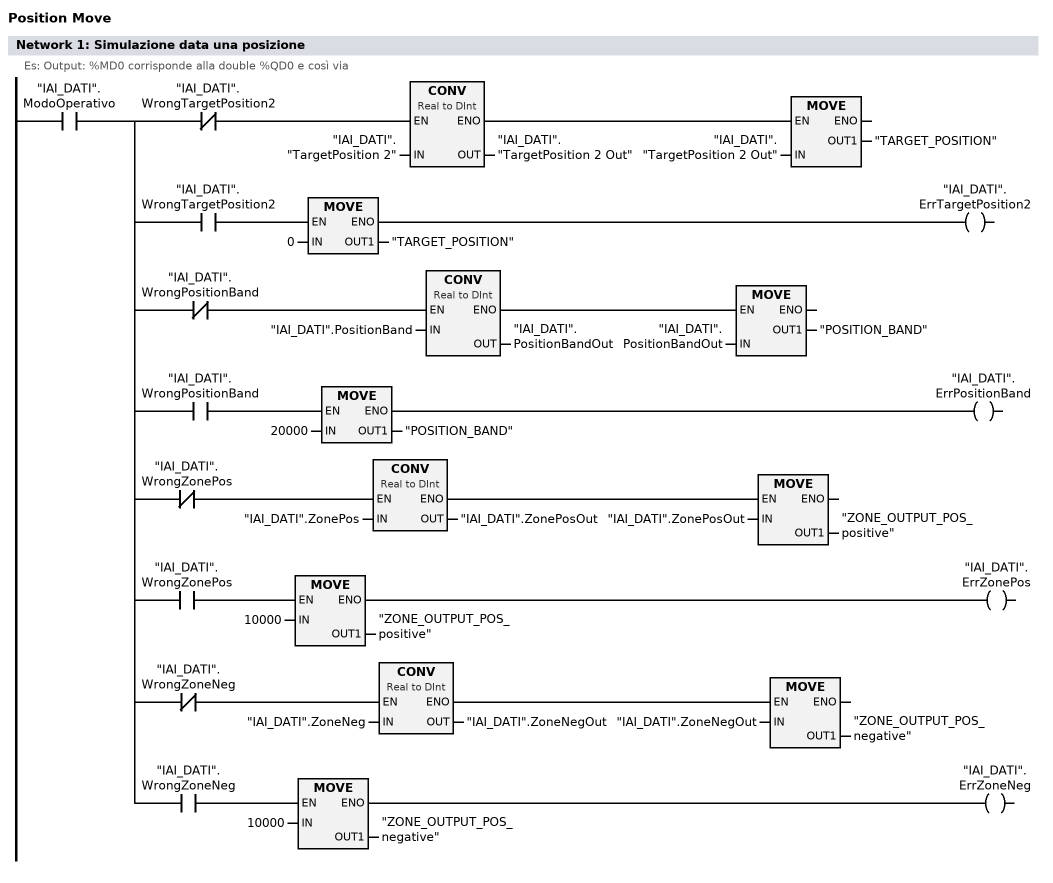
   RUNG wire#powerrail
      Contact( "IAI_DATI".ModoOperativo )
      wire#w1
      I_Contact( "IAI_DATI".WrongTargetPosition2 )
      { S7_Templates := "[SrcType := Real, DestType := DInt]" } Convert(in := "IAI_DATI"."TargetPosition 2", out => "IAI_DATI"."TargetPosition 2 Out")
      Move(in := "IAI_DATI"."TargetPosition 2 Out", out1 => "TARGET_POSITION")
   END_RUNG
   RUNG wire#w1
      Contact( "IAI_DATI".WrongTargetPosition2 )
      Move(in := 0, out1 => "TARGET_POSITION")
      Coil( "IAI_DATI".ErrTargetPosition2 )
   END_RUNG
   RUNG wire#w1
      I_Contact( "IAI_DATI".WrongPositionBand )
      { S7_Templates := "[SrcType := Real, DestType := DInt]" } Convert(in := "IAI_DATI".PositionBand, out => "IAI_DATI".PositionBandOut)
      Move(in := "IAI_DATI".PositionBandOut, out1 => "POSITION_BAND")
   END_RUNG
   RUNG wire#w1
      Contact( "IAI_DATI".WrongPositionBand )
      Move(in := 20000, out1 => "POSITION_BAND")
      Coil( "IAI_DATI".ErrPositionBand )
   END_RUNG
   RUNG wire#w1
      I_Contact( "IAI_DATI".WrongZonePos )
      { S7_Templates := "[SrcType := Real, DestType := DInt]" } Convert(in := "IAI_DATI".ZonePos, out => "IAI_DATI".ZonePosOut)
      Move(in := "IAI_DATI".ZonePosOut, out1 => "ZONE_OUTPUT_POS_positive")
   END_RUNG
   RUNG wire#w1
      Contact( "IAI_DATI".WrongZonePos )
      Move(in := 10000, out1 => "ZONE_OUTPUT_POS_positive")
      Coil( "IAI_DATI".ErrZonePos )
   END_RUNG
   RUNG wire#w1
      I_Contact( "IAI_DATI".WrongZoneNeg )
      { S7_Templates := "[SrcType := Real, DestType := DInt]" } Convert(in := "IAI_DATI".ZoneNeg, out => "IAI_DATI".ZoneNegOut)
      Move(in := "IAI_DATI".ZoneNegOut, out1 => "ZONE_OUTPUT_POS_negative")
   END_RUNG
   RUNG wire#w1
      Contact( "IAI_DATI".WrongZoneNeg )
      Move(in := 10000, out1 => "ZONE_OUTPUT_POS_negative")
      Coil( "IAI_DATI".ErrZoneNeg )
   END_RUNG
   // the same network as SCL:
   IF "IAI_DATI".ModoOperativo AND NOT "IAI_DATI".WrongTargetPosition2 THEN
       "IAI_DATI"."TargetPosition 2 Out" := REAL_TO_DINT("IAI_DATI"."TargetPosition 2");
       "TARGET_POSITION" := "IAI_DATI"."TargetPosition 2 Out";
   END_IF;
   #_w1 := "IAI_DATI".ModoOperativo AND "IAI_DATI".WrongTargetPosition2;
   IF #_w1 THEN "TARGET_POSITION" := 0; END_IF;
   "IAI_DATI".ErrTargetPosition2 := #_w1;
   IF "IAI_DATI".ModoOperativo AND NOT "IAI_DATI".WrongPositionBand THEN
       "IAI_DATI".PositionBandOut := REAL_TO_DINT("IAI_DATI".PositionBand);
       "POSITION_BAND" := "IAI_DATI".PositionBandOut;
   END_IF;
   #_w2 := "IAI_DATI".ModoOperativo AND "IAI_DATI".WrongPositionBand;
   IF #_w2 THEN "POSITION_BAND" := 20000; END_IF;
   "IAI_DATI".ErrPositionBand := #_w2;
   IF "IAI_DATI".ModoOperativo AND NOT "IAI_DATI".WrongZonePos THEN
       "IAI_DATI".ZonePosOut := REAL_TO_DINT("IAI_DATI".ZonePos);
       "ZONE_OUTPUT_POS_positive" := "IAI_DATI".ZonePosOut;
   END_IF;
   #_w3 := "IAI_DATI".ModoOperativo AND "IAI_DATI".WrongZonePos;
   IF #_w3 THEN "ZONE_OUTPUT_POS_positive" := 10000; END_IF;
   "IAI_DATI".ErrZonePos := #_w3;
   IF "IAI_DATI".ModoOperativo AND NOT "IAI_DATI".WrongZoneNeg THEN
       "IAI_DATI".ZoneNegOut := REAL_TO_DINT("IAI_DATI".ZoneNeg);
       "ZONE_OUTPUT_POS_negative" := "IAI_DATI".ZoneNegOut;
   END_IF;
   #_w4 := "IAI_DATI".ModoOperativo AND "IAI_DATI".WrongZoneNeg;
   IF #_w4 THEN "ZONE_OUTPUT_POS_negative" := 10000; END_IF;
   "IAI_DATI".ErrZoneNeg := #_w4;
END_REGION
END_FUNCTION_BLOCK

FUNCTION_BLOCK "Speed Move"   // FB4, LAD
TITLE = Speed Move
{ S7_Optimized_Access := 'TRUE' }
AUTHOR : Valentino-Fabbri
VERSION : 0.1
   VAR_TEMP   // added for the SCL form of the ladder/FBD networks
      _w1 : Bool;
      _w2 : Bool;
      _w3 : Bool;
      _w4 : Bool;
   END_VAR
BEGIN

REGION Network 1: Simulazione in Jog
   // Es: Output: %MD8 corrisponde alla double %QD8 e così via
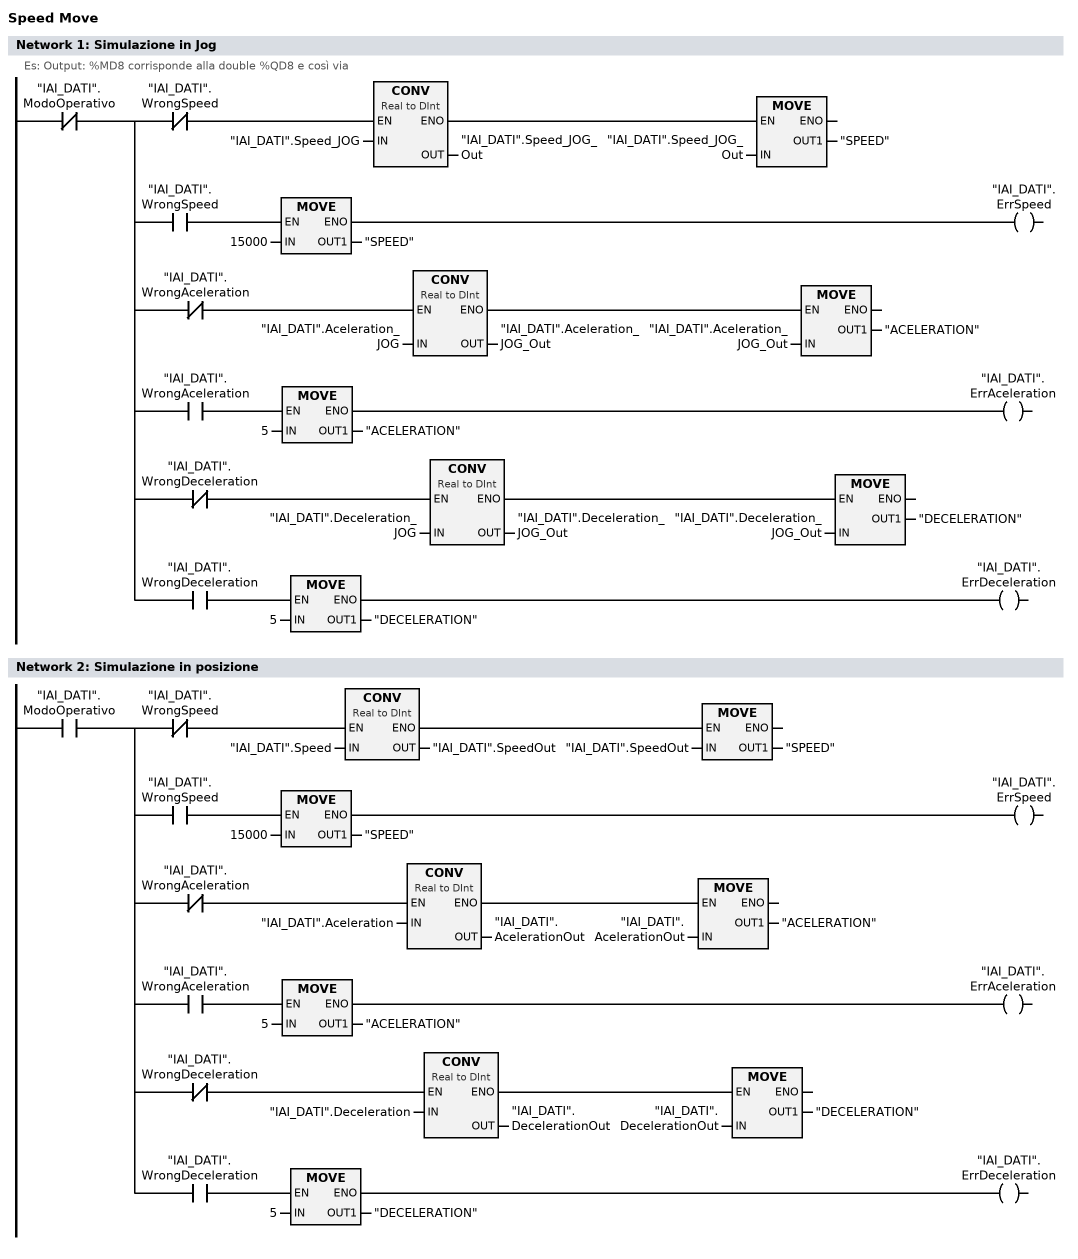
   RUNG wire#powerrail
      I_Contact( "IAI_DATI".ModoOperativo )
      wire#w1
      I_Contact( "IAI_DATI".WrongSpeed )
      { S7_Templates := "[SrcType := Real, DestType := DInt]" } Convert(in := "IAI_DATI".Speed_JOG, out => "IAI_DATI".Speed_JOG_Out)
      Move(in := "IAI_DATI".Speed_JOG_Out, out1 => "SPEED")
   END_RUNG
   RUNG wire#w1
      Contact( "IAI_DATI".WrongSpeed )
      Move(in := 15000, out1 => "SPEED")
      Coil( "IAI_DATI".ErrSpeed )
   END_RUNG
   RUNG wire#w1
      I_Contact( "IAI_DATI".WrongAceleration )
      { S7_Templates := "[SrcType := Real, DestType := DInt]" } Convert(in := "IAI_DATI".Aceleration_JOG, out => "IAI_DATI".Aceleration_JOG_Out)
      Move(in := "IAI_DATI".Aceleration_JOG_Out, out1 => "ACELERATION")
   END_RUNG
   RUNG wire#w1
      Contact( "IAI_DATI".WrongAceleration )
      Move(in := 5, out1 => "ACELERATION")
      Coil( "IAI_DATI".ErrAceleration )
   END_RUNG
   RUNG wire#w1
      I_Contact( "IAI_DATI".WrongDeceleration )
      { S7_Templates := "[SrcType := Real, DestType := DInt]" } Convert(in := "IAI_DATI".Deceleration_JOG, out => "IAI_DATI".Deceleration_JOG_Out)
      Move(in := "IAI_DATI".Deceleration_JOG_Out, out1 => "DECELERATION")
   END_RUNG
   RUNG wire#w1
      Contact( "IAI_DATI".WrongDeceleration )
      Move(in := 5, out1 => "DECELERATION")
      Coil( "IAI_DATI".ErrDeceleration )
   END_RUNG
   // the same network as SCL:
   #_w1 := NOT "IAI_DATI".ModoOperativo;
   IF #_w1 AND NOT "IAI_DATI".WrongSpeed THEN
       "IAI_DATI".Speed_JOG_Out := REAL_TO_DINT("IAI_DATI".Speed_JOG);
       "SPEED" := "IAI_DATI".Speed_JOG_Out;
   END_IF;
   #_w2 := #_w1 AND "IAI_DATI".WrongSpeed;
   IF #_w2 THEN "SPEED" := 15000; END_IF;
   "IAI_DATI".ErrSpeed := #_w2;
   IF #_w1 AND NOT "IAI_DATI".WrongAceleration THEN
       "IAI_DATI".Aceleration_JOG_Out := REAL_TO_DINT("IAI_DATI".Aceleration_JOG);
       "ACELERATION" := "IAI_DATI".Aceleration_JOG_Out;
   END_IF;
   #_w3 := #_w1 AND "IAI_DATI".WrongAceleration;
   IF #_w3 THEN "ACELERATION" := 5; END_IF;
   "IAI_DATI".ErrAceleration := #_w3;
   IF #_w1 AND NOT "IAI_DATI".WrongDeceleration THEN
       "IAI_DATI".Deceleration_JOG_Out := REAL_TO_DINT("IAI_DATI".Deceleration_JOG);
       "DECELERATION" := "IAI_DATI".Deceleration_JOG_Out;
   END_IF;
   #_w4 := #_w1 AND "IAI_DATI".WrongDeceleration;
   IF #_w4 THEN "DECELERATION" := 5; END_IF;
   "IAI_DATI".ErrDeceleration := #_w4;
END_REGION

REGION Network 2: Simulazione in posizione
   RUNG wire#powerrail
      Contact( "IAI_DATI".ModoOperativo )
      wire#w1
      I_Contact( "IAI_DATI".WrongSpeed )
      { S7_Templates := "[SrcType := Real, DestType := DInt]" } Convert(in := "IAI_DATI".Speed, out => "IAI_DATI".SpeedOut)
      Move(in := "IAI_DATI".SpeedOut, out1 => "SPEED")
   END_RUNG
   RUNG wire#w1
      Contact( "IAI_DATI".WrongSpeed )
      Move(in := 15000, out1 => "SPEED")
      Coil( "IAI_DATI".ErrSpeed )
   END_RUNG
   RUNG wire#w1
      I_Contact( "IAI_DATI".WrongAceleration )
      { S7_Templates := "[SrcType := Real, DestType := DInt]" } Convert(in := "IAI_DATI".Aceleration, out => "IAI_DATI".AcelerationOut)
      Move(in := "IAI_DATI".AcelerationOut, out1 => "ACELERATION")
   END_RUNG
   RUNG wire#w1
      Contact( "IAI_DATI".WrongAceleration )
      Move(in := 5, out1 => "ACELERATION")
      Coil( "IAI_DATI".ErrAceleration )
   END_RUNG
   RUNG wire#w1
      I_Contact( "IAI_DATI".WrongDeceleration )
      { S7_Templates := "[SrcType := Real, DestType := DInt]" } Convert(in := "IAI_DATI".Deceleration, out => "IAI_DATI".DecelerationOut)
      Move(in := "IAI_DATI".DecelerationOut, out1 => "DECELERATION")
   END_RUNG
   RUNG wire#w1
      Contact( "IAI_DATI".WrongDeceleration )
      Move(in := 5, out1 => "DECELERATION")
      Coil( "IAI_DATI".ErrDeceleration )
   END_RUNG
   // the same network as SCL:
   IF "IAI_DATI".ModoOperativo AND NOT "IAI_DATI".WrongSpeed THEN
       "IAI_DATI".SpeedOut := REAL_TO_DINT("IAI_DATI".Speed);
       "SPEED" := "IAI_DATI".SpeedOut;
   END_IF;
   #_w1 := "IAI_DATI".ModoOperativo AND "IAI_DATI".WrongSpeed;
   IF #_w1 THEN "SPEED" := 15000; END_IF;
   "IAI_DATI".ErrSpeed := #_w1;
   IF "IAI_DATI".ModoOperativo AND NOT "IAI_DATI".WrongAceleration THEN
       "IAI_DATI".AcelerationOut := REAL_TO_DINT("IAI_DATI".Aceleration);
       "ACELERATION" := "IAI_DATI".AcelerationOut;
   END_IF;
   #_w2 := "IAI_DATI".ModoOperativo AND "IAI_DATI".WrongAceleration;
   IF #_w2 THEN "ACELERATION" := 5; END_IF;
   "IAI_DATI".ErrAceleration := #_w2;
   IF "IAI_DATI".ModoOperativo AND NOT "IAI_DATI".WrongDeceleration THEN
       "IAI_DATI".DecelerationOut := REAL_TO_DINT("IAI_DATI".Deceleration);
       "DECELERATION" := "IAI_DATI".DecelerationOut;
   END_IF;
   #_w3 := "IAI_DATI".ModoOperativo AND "IAI_DATI".WrongDeceleration;
   IF #_w3 THEN "DECELERATION" := 5; END_IF;
   "IAI_DATI".ErrDeceleration := #_w3;
END_REGION
END_FUNCTION_BLOCK

FUNCTION_BLOCK "DoubleTapButton2"   // FB5, LAD
{ S7_Optimized_Access := 'TRUE' }
VERSION : 0.1
   VAR_INPUT
      Button : Bool;
   END_VAR
   VAR_IN_OUT
      Out : Bool;
      Set : Bool;
      Reset : Bool;
      ResetCTU : Bool;
      IEC_Counter : IEC_COUNTER;
   END_VAR
   VAR_TEMP
      MLB : Int;
   END_VAR
BEGIN

REGION Network 1: Conta click
   // Conto i due fronti dei click e resetto arrivato al secondo
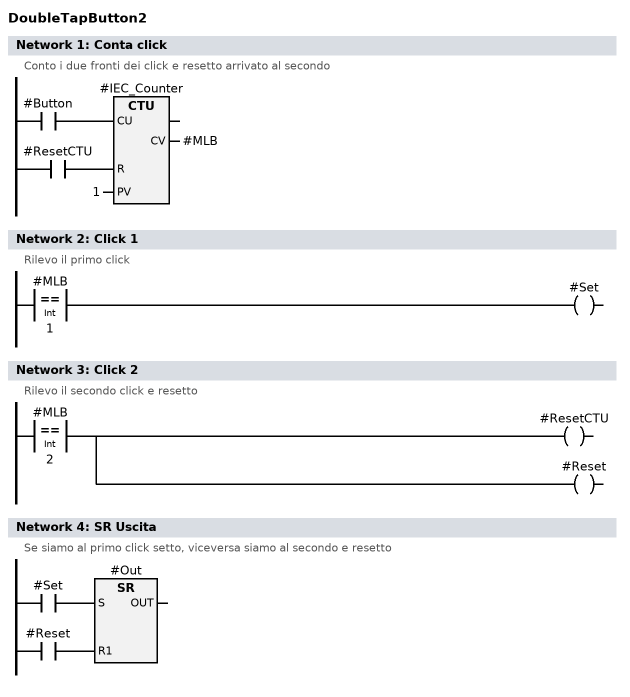
   #IEC_Counter.CTU(CU := #Button, R := #ResetCTU, PV := 1, CV => #MLB);
END_REGION

REGION Network 2: Click 1
   // Rilevo il primo click
   RUNG wire#powerrail
      { S7_Templates := "SrcType := Int" } EQ_Contact(in1 := #MLB, in2 := 1)
      Coil( #Set )
   END_RUNG
   // the same network as SCL:
   #Set := #MLB = 1;
END_REGION

REGION Network 3: Click 2
   // Rilevo il secondo click e resetto
   RUNG wire#powerrail
      { S7_Templates := "SrcType := Int" } EQ_Contact(in1 := #MLB, in2 := 2)
      wire#w1
      Coil( #ResetCTU )
   END_RUNG
   RUNG wire#w1
      Coil( #Reset )
   END_RUNG
   // the same network as SCL:
   #ResetCTU := #MLB = 2;
   #Reset := #ResetCTU;
END_REGION

REGION Network 4: SR Uscita
   // Se siamo al primo click setto, viceversa siamo al secondo e resetto
   RUNG wire#powerrail
      Contact( #Set )
      S_SR(operand := #Out, r1 := wire#w1)
   END_RUNG
   RUNG wire#powerrail
      Contact( #Reset )
   END_RUNG wire#w1
   // the same network as SCL:
   IF #Set THEN
       #Out := TRUE;   // SR flip-flop
   END_IF;
   IF #Reset THEN #Out := FALSE; END_IF;
END_REGION
END_FUNCTION_BLOCK

FUNCTION_BLOCK "CollisionMovement"   // FB6, LAD
TITLE = CollisionMovement
{ S7_Optimized_Access := 'TRUE' }
AUTHOR : Valentino-Fabbri
VERSION : 0.1
   VAR_INPUT
      Start : Bool;
      MeasureValue : Real;
      ErrorTimeOut : Time;
      PositionEnd : Bool;
   END_VAR
   VAR_OUTPUT
      EnableLog : Bool;
      ReadError : Bool;
   END_VAR
   VAR_IN_OUT
      EnableRec : Bool;
      IEC_TP_ReadError : TP_TIME;
   END_VAR
BEGIN

REGION Network 1: Attivo la lettura
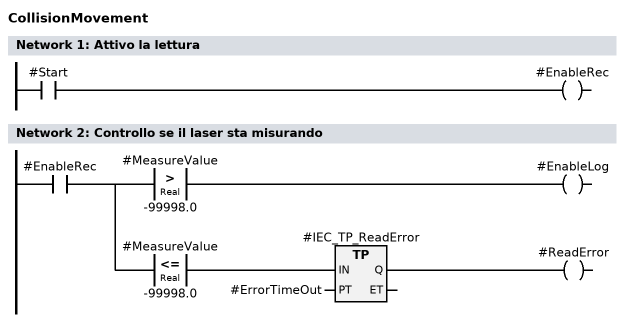
   RUNG wire#powerrail
      Contact( #Start )
      Coil( #EnableRec )
   END_RUNG
   // the same network as SCL:
   #EnableRec := #Start;
END_REGION

REGION Network 2: Controllo se il laser sta misurando
   #EnableLog := #EnableRec AND (#MeasureValue > (-99998.0));
   #IEC_TP_ReadError(IN := #EnableRec AND (#MeasureValue <= (-99998.0)), PT := #ErrorTimeOut);   // TP
   #ReadError := #IEC_TP_ReadError.Q;
END_REGION
END_FUNCTION_BLOCK

FUNCTION_BLOCK "Input"   // FB7, LAD
TITLE = Assegno Input
{ S7_Optimized_Access := 'TRUE' }
AUTHOR : Valentino-Fabbri
VERSION : 0.1
BEGIN

REGION Network 1: Posizione completata
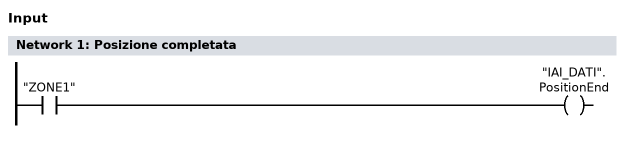
   RUNG wire#powerrail
      Contact( "ZONE1" )
      Coil( "IAI_DATI".PositionEnd )
   END_RUNG
   // the same network as SCL:
   "IAI_DATI".PositionEnd := "ZONE1";
END_REGION
END_FUNCTION_BLOCK

// folder: Funzioni

FUNCTION "RND" : Void   // FC1, SCL
TITLE = Random
{ S7_Optimized_Access := 'TRUE' }
AUTHOR : Valentino-Fabbri
VERSION : 0.1
   VAR_INPUT
      Seed : Word;
      Restart : Bool;
   END_VAR
   VAR_OUTPUT
      Rand_Num : Word;
   END_VAR
   VAR_TEMP
      wRandomVar : Word;
      aRandomVar : Array[0..15] of Bool;
   END_VAR
BEGIN
   #wRandomVar := 751;

   IF #Restart = TRUE THEN
       #wRandomVar := #Seed;
   ELSE
       #aRandomVar[6] := 0;
       #aRandomVar[7] := 0;
       #wRandomVar := DINT_TO_WORD(WORD_TO_DINT(#wRandomVar) + WORD_TO_DINT(#wRandomVar));
       #aRandomVar[8] := #aRandomVar[14] XOR #aRandomVar[5];
       #Rand_Num := #wRandomVar;
   END_IF;
END_FUNCTION

FUNCTION "DoubleTapButton" : Void   // FC2, LAD
TITLE = Double Tap
{ S7_Optimized_Access := 'TRUE' }
AUTHOR : Valentino-Fabbri
VERSION : 0.1
   VAR_INPUT
      Button : Bool;
   END_VAR
   VAR_IN_OUT
      Out : Bool;
      Set : Bool;
      Reset : Bool;
      ResetCTU : Bool;
      IEC_Counter : IEC_COUNTER;
   END_VAR
   VAR_TEMP
      MLB : Int;
   END_VAR
BEGIN

REGION Network 1: Conta click
   // Conto i due fronti dei click e resetto arrivato al secondo
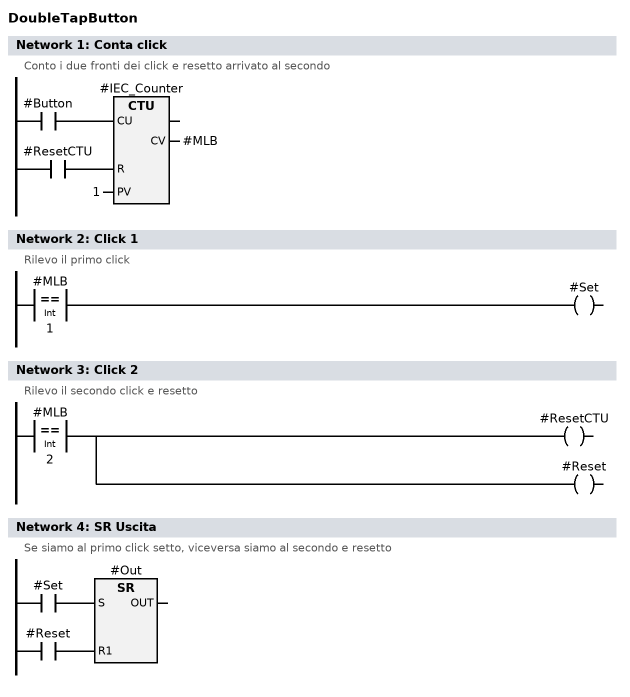
   #IEC_Counter.CTU(CU := #Button, R := #ResetCTU, PV := 1, CV => #MLB);
END_REGION

REGION Network 2: Click 1
   // Rilevo il primo click
   RUNG wire#powerrail
      { S7_Templates := "SrcType := Int" } EQ_Contact(in1 := #MLB, in2 := 1)
      Coil( #Set )
   END_RUNG
   // the same network as SCL:
   #Set := #MLB = 1;
END_REGION

REGION Network 3: Click 2
   // Rilevo il secondo click e resetto
   RUNG wire#powerrail
      { S7_Templates := "SrcType := Int" } EQ_Contact(in1 := #MLB, in2 := 2)
      wire#w1
      Coil( #ResetCTU )
   END_RUNG
   RUNG wire#w1
      Coil( #Reset )
   END_RUNG
   // the same network as SCL:
   #ResetCTU := #MLB = 2;
   #Reset := #ResetCTU;
END_REGION

REGION Network 4: SR Uscita
   // Se siamo al primo click setto, viceversa siamo al secondo e resetto
   RUNG wire#powerrail
      Contact( #Set )
      S_SR(operand := #Out, r1 := wire#w1)
   END_RUNG
   RUNG wire#powerrail
      Contact( #Reset )
   END_RUNG wire#w1
   // the same network as SCL:
   IF #Set THEN
       #Out := TRUE;   // SR flip-flop
   END_IF;
   IF #Reset THEN #Out := FALSE; END_IF;
END_REGION
END_FUNCTION

(* ===== HMI "HMI_RT_1" =====
system functions are stored by id; their names below are inferred from use
connection "HMI_Collegamento_1": ETHERNET, S7_1500_OMS

HMI tags "Tabella delle variabili standard"
   "IAI_DATI_PositionBand" : Real = PLC IAI_DATI.PositionBand, 1 s
      on AboveUpperLimit: "ShowError"('IAI_DATI_PositionBand', 'IAI_DATI_WrongPositionBand', "IAI_DATI_PositionBandLowLimit", "IAI_DATI_PositionBandHighLimit")
      on BelowLowerLimit: "ShowError"('IAI_DATI_PositionBand', 'IAI_DATI_WrongPositionBand', "IAI_DATI_PositionBandLowLimit", "IAI_DATI_PositionBandHighLimit")
   "IAI_DATI_Speed" : Real = PLC IAI_DATI.Speed, 1 s
      on AboveUpperLimit: "ShowError"('IAI_DATI_Speed', 'IAI_DATI.WrongSpeed', "IAI_DATI_SpeedLowLimit", "IAI_DATI_SpeedHighLimit")
      on BelowLowerLimit: "ShowError"('IAI_DATI_Speed', 'IAI_DATI.WrongSpeed', "IAI_DATI_SpeedLowLimit", "IAI_DATI_SpeedHighLimit")
   "IAI_DATI_Aceleration" : Real = PLC IAI_DATI.Aceleration, 1 s
      on AboveUpperLimit: "ShowError"('IAI_DATI_Aceleration', 'IAI_DATI.WrongAceleration', "IAI_DATI_AcelerationLowLimit", "IAI_DATI_AcelerationHighLimit")
      on BelowLowerLimit: "ShowError"('IAI_DATI_Aceleration', 'IAI_DATI.WrongAceleration', "IAI_DATI_AcelerationLowLimit", "IAI_DATI_AcelerationHighLimit")
   "IAI_DATI_Deceleration" : Real = PLC IAI_DATI.Deceleration, 1 s
      on AboveUpperLimit: "ShowError"('IAI_DATI_Deceleration', 'IAI_DATI.WrongDeceleration', "IAI_DATI_DecelerationLowLimit", "IAI_DATI_DecelerationHighLimit")
      on BelowLowerLimit: "ShowError"('IAI_DATI_Deceleration', 'IAI_DATI.WrongDeceleration', "IAI_DATI_DecelerationLowLimit", "IAI_DATI_DecelerationHighLimit")
   "M_SON_AXIS" : Bool = PLC M_SON_AXIS AT %M100.0, 1 s
   "M_STR_AXIS" : Bool = PLC M_STR_AXIS AT %M100.1, 1 s
   "M_DSTR_ON" : Bool = PLC M_DSTR_ON AT %M100.2, 1 s
   "RECORD_IL1000" : DInt = PLC Keyence_DATI.Record AT %MD215, 1 s
   "M_RETURN_HOME" : Bool = PLC M_RETURN_HOME AT %M400.0, 1 s
   "IAI_DATI_ZonePos" : Real = PLC IAI_DATI.ZonePos, 1 s
      on AboveUpperLimit: "ShowError"('IAI_DATI_ZonePos', 'IAI_DATI.WrongZonePos', "IAI_DATI_ZonePosLowLimit", "IAI_DATI_ZonePosHighLimit")
      on BelowLowerLimit: "ShowError"('IAI_DATI_ZonePos', 'IAI_DATI.WrongZonePos', "IAI_DATI_ZonePosLowLimit", "IAI_DATI_ZonePosHighLimit")
   "IAI_DATI_ZonNeg" : Real = PLC IAI_DATI.ZoneNeg, 1 s
      on AboveUpperLimit: "ShowError"('IAI_DATI_ZoneNeg', 'IAI_DATI.WrongZoneNeg', "IAI_DATI_ZoneNegLowLimit", "IAI_DATI_ZoneNegHighLimit")
      on BelowLowerLimit: "ShowError"('IAI_DATI_ZoneNeg', 'IAI_DATI.WrongZoneNeg', "IAI_DATI_ZoneNegLowLimit", "IAI_DATI_ZoneNegHighLimit")
   "RES" : Bool = PLC RES AT %Q31.3, 1 s
   "JOGneg" : Bool = PLC JOGneg AT %Q31.7, 1 s
   "JOGpos" : Bool = PLC JOGpos AT %Q30.0, 1 s
   "IL_100_ST" : Bool = PLC IL_100_ST AT %M100.6, 1 s
   "M_RESET_ALLARM" : Bool = PLC M_RESET_ALLARM AT %M100.5, 1 s
   "M_JOG_POS" : Bool = PLC M_JOG_POS AT %M100.3, 1 s
   "M_JOG_NEG" : Bool = PLC M_JOG_NEG AT %M100.4, 1 s
   "IAI_DATI_TargetPosition 1" : DInt = PLC IAI_DATI."TargetPosition 1" AT %DB1.DBX0.0, 1 s
   "IAI_DATI_TargetPosition 2" : Real = PLC IAI_DATI."TargetPosition 2" AT %DB1.DBD0, 1 s
      on AboveUpperLimit: "ShowError"('IAI_DATI_TargetPosition 2', 'IAI_DATI.WrongTargetPosition2', "IAI_DATI_TargetPosition2LowLimit", "IAI_DATI_TargetPosition2HighLimit")
      on BelowLowerLimit: "ShowError"('IAI_DATI_TargetPosition 2', 'IAI_DATI.WrongTargetPosition2', "IAI_DATI_TargetPosition2LowLimit", "IAI_DATI_TargetPosition2HighLimit")
   "IAI_DATI_Speed_JOG" : Real = PLC IAI_DATI.Speed_JOG AT %DB1.DBD0, 1 s
      on AboveUpperLimit: "ShowError"('IAI_DATI_Speed_Jog', 'IAI_DATI.WrongSpeed', "IAI_DATI_SpeedLowLimit", "IAI_DATI_SpeedHighLimit")
   "IAI_DATI_Aceleration_JOG" : Real = PLC IAI_DATI.Aceleration_JOG AT %DB1.DBD0, 1 s
      on AboveUpperLimit: "ShowError"('IAI_DATI_Aceleration_JOG', 'IAI_DATI.WrongAceleration', "IAI_DATI_AcelerationLowLimit", "IAI_DATI_AcelerationHighLimit")
      on BelowLowerLimit: "ShowError"('IAI_DATI_Aceleration_Jog', 'IAI_DATI.WrongAceleration', "IAI_DATI_AcelerationLowLimit", "IAI_DATI_AcelerationHighLimit")
   "IAI_DATI_Deceleration_JOG" : Real = PLC IAI_DATI.Deceleration_JOG AT %DB1.DBD0, 1 s
      on AboveUpperLimit: "ShowError"('IAI_DATI_Deceleration_Jog', 'IAI_DATI.WrongDeceleration', "IAI_DATI_DecelerationLowLimit", "IAI_DATI_DecelerationHighLimit")
      on BelowLowerLimit: "ShowError"('IAI_DATI_Deceleration_Jog', 'IAI_DATI.WrongDeceleration', "IAI_DATI_DecelerationLowLimit", "IAI_DATI_DecelerationHighLimit")
   "IAI_DATI_ActualPosition" : Real = PLC IAI_DATI.ActualPosition AT %DB1.DBD0, 100 ms
   "Keyence_DATI_MeasureValue" : Real = PLC Keyence_DATI.MeasureValue AT %DB1.DBD0, 100 ms
   "IAI_DATI_ModoOperativo" : Bool = PLC IAI_DATI.ModoOperativo AT %DB1.DBD0, 1 s
   "Rugosimetro_Ra" : Real = PLC Rugosimetro.Ra, 1 s
   "SQL_ChangeValue" : Bool = PLC SQL.ChangeValue, 100 ms
      on ChangeValue: "ReportOffline"(); "CheckCollision"()
   "SelectOPMode" : Bool = PLC SelectOPMode AT %M10.0, 1 s
   "SQL_SendValue" : Time = PLC SQL.SendValue, 1 s
   "Keyence_DATI_ARLM_IL_1000" : Int = PLC Keyence_DATI.ARLM_IL_1000, 1 s
   "Rnd_Restart" : Bool = PLC Rnd_Restart AT %M20.0, 1 s
   "Restart_Sim" : Bool = PLC Restart_Sim AT %M30.0, 1 s
   "Keyence_DATI_Request" : Bool = PLC Keyence_DATI.Request, 1 s
   "REQ_IL1000" : Bool = PLC REQ_IL1000 AT %M500.0, 1 s
   "Keyence_DATI_IsBusy" : Bool = PLC Keyence_DATI.IsBusy, 1 s
   "Keyence_DATI_IsValid" : Bool = PLC Keyence_DATI.IsValid, 1 s
   "Keyence_DATI_IsError" : Bool = PLC Keyence_DATI.IsError, 1 s
   "SQL_SetName" : String[10] = PLC SQL.SetName, 1 s
   "SQL_SendFile" : Int = PLC SQL.SendFile AT %DB1.DBX0.0, 100 ms
      on AboveUpperLimit: "Report"()
   "SQL_BtnSend" : Bool = PLC SQL.BtnSend, 1 s
   "SQL_CheckState" : Int = PLC SQL.CheckState AT %DB1.DBX0.0, 100 ms
   "Simulation_HighMax" : DWord = PLC Simulation.HighMax, 1 s
   "Simulation_PositionMax" : DWord = PLC Simulation.PositionMax, 1 s
   "Simulation_SimuTimeIn" : Time = PLC Simulation.SimuTimeIn, 1 s
   "Simulation_SimuTimeOut" : Time = PLC Simulation.SimuTimeOut, 1 s
   "SQL_CTUAlt" : Real = PLC SQL.CTUAlt, 100 ms
   "SQL_CTUPos" : Real = PLC SQL.CTUPos, 100 ms
   "Keyence_DATI_Activate" : Bool = PLC Keyence_DATI.Activate, 1 s
   "RawPosition" : DWord = PLC RawPosition AT %ID0, 1 s
   "IAI_DATI_ErrPositionBand" : Bool = PLC IAI_DATI.ErrPositionBand, 1 s
   "IAI_DATI_ErrSpeed" : Bool = PLC IAI_DATI.ErrSpeed, 1 s
   "IAI_DATI_ErrDeceleration" : Bool = PLC IAI_DATI.ErrDeceleration, 1 s
   "IAI_DATI_ErrAceleration" : Bool = PLC IAI_DATI.ErrAceleration, 1 s
   "IAI_DATI_ErrZonePos" : Bool = PLC IAI_DATI.ErrZonePos, 1 s
   "IAI_DATI_ErrZoneNeg" : Bool = PLC IAI_DATI.ErrZoneNeg, 1 s
   "IAI_DATI_WrongPositionBand" : Bool = PLC IAI_DATI.WrongPositionBand, 1 s
   "IAI_DATI_PositionBandHighLimit" : Real = PLC IAI_DATI.PositionBandHighLimit, 1 s
   "IAI_DATI_PositionBandLowLimit" : Real = PLC IAI_DATI.PositionBandLowLimit, 1 s
   "IAI_DATI_SpeedHighLimit" : Real = PLC IAI_DATI.SpeedHighLimit, 1 s
   "IAI_DATI_SpeedLowLimit" : Real = PLC IAI_DATI.SpeedLowLimit, 1 s
   "IAI_DATI_AcelerationHighLimit" : Real = PLC IAI_DATI.AcelerationHighLimit, 1 s
   "IAI_DATI_AcelerationLowLimit" : Real = PLC IAI_DATI.AcelerationLowLimit, 1 s
   "IAI_DATI.WrongTargetPosition2" : Bool = PLC IAI_DATI.WrongTargetPosition2 AT %DB1.DBD0, 1 s
   "IAI_DATI.WrongZonePos" : Bool = PLC IAI_DATI.WrongZonePos AT %DB1.DBX0.0, 1 s
   "IAI_DATI.WrongZoneNeg" : Bool = PLC IAI_DATI.WrongZoneNeg AT %DB1.DBX0.0, 1 s
   "IAI_DATI.WrongSpeed" : Bool = PLC IAI_DATI.WrongSpeed AT %DB1.DBX0.0, 1 s
   "IAI_DATI.WrongAceleration" : Bool = PLC IAI_DATI.WrongAceleration AT %DB1.DBX0.0, 1 s
   "IAI_DATI.WrongDeceleration" : Bool = PLC IAI_DATI.WrongDeceleration AT %DB1.DBX0.0, 1 s
   "IAI_DATI_TargetPosition2HighLimit" : Real = PLC IAI_DATI.TargetPosition2HighLimit, 1 s
   "IAI_DATI_TargetPosition2LowLimit" : Real = PLC IAI_DATI.TargetPosition2LowLimit, 1 s
   "IAI_DATI_ZonePosHighLimit" : Real = PLC IAI_DATI.ZonePosHighLimit, 1 s
   "IAI_DATI_ZonePosLowLimit" : Real = PLC IAI_DATI.ZonePosLowLimit, 1 s
   "IAI_DATI_ZoneNegHighLimit" : Real = PLC IAI_DATI.ZoneNegHighLimit, 1 s
   "IAI_DATI_ZoneNegLowLimit" : Real = PLC IAI_DATI.ZoneNegLowLimit, 1 s
   "Keyence_DATI_ReadError" : Bool = PLC Keyence_DATI.ReadError, 1 s
   "Keyence_DATI.ReadError" : Bool = PLC Keyence_DATI.ReadError AT %DB1.DBX0.0, 1 s
      on ChangeValue: "CheckCollision"()
   "IAI_DATI_ErrTargetPosition2" : Bool = PLC IAI_DATI.ErrTargetPosition2, 1 s
   "IAI_DATI_DecelerationLowLimit" : Real = PLC IAI_DATI.DecelerationLowLimit, 1 s
   "IAI_DATI_DecelerationHighLimit" : Real = PLC IAI_DATI.DecelerationHighLimit, 1 s

discrete alarms
   1: 'Si è verificata un anomalia nella lettura del componente IL_1000', class Errors, trigger "Keyence_DATI_ARLM_IL_1000" bit 1

text list "Jog/Auto": 0 'Jog'; 1 'Auto'

text list "Pos/Neg": -2 'Neg'; 2 'Pos'; 0 'Off'

text list "SQLState": 0 'Offline'; 1 'Online'

text list "On/Off": 0 'Off'; 1 'On'

text list "Ok/Ko": 0 'Ko'; 1 'Ok'

text list "Read_Prof": 0 'Disabilitato'; 1 'Abilitato'

screen "Rugosimetro" 480x272, template "Modello_1"
   Softkey "Softkey_F2" at 0,0 size 0x0
      on KeyDown: SetBit("M_RESET_ALLARM")
      on KeyUp: ResetBit("M_RESET_ALLARM")
   Softkey "Softkey_F3" at 0,0 size 0x0
      on KeyDown: SetBit("IL_100_ST")
      on KeyUp: ResetBit("IL_100_ST")
   Softkey "Softkey_F4" at 0,0 size 0x0
      on KeyDown: SetBit("M_JOG_POS")
      on KeyUp: ResetBit("M_JOG_POS")
   Button "Pulsante_4" at 360,140 size 96x30; TextOff 'Start'
      on Press: SetBit("M_DSTR_ON")
      on Release: ResetBit("M_DSTR_ON")
   Button "Pulsante_1" at 360,70 size 96x30; TextOff 'Home'
      on Release: ResetBit("M_RETURN_HOME")
      on Press: SetBit("M_RETURN_HOME")
   TextField "Casella di testo_4" at 6,75 size 133x20; Text 'Posizione attuale'
   TextField "Casella di testo_7" at 6,181 size 65x20; Text 'Velocità'
   TextField "Casella di testo_6" at 6,145 size 121x20; Text 'Pos. desiderata'
   IOField "Campo I/O_2" at 227,140 size 96x30; FormatPattern s99999
      ProcessValue <- "IAI_DATI_TargetPosition 2"
      Appearance <- "IAI_DATI_ErrTargetPosition2"
   TextField "Casella di testo_1" at 6,110 size 156x20; Text 'Rugosità media (Ra)'
   IOField "Campo I/O_1" at 227,70 size 96x30; FormatPattern s999.99999
      ProcessValue <- "IAI_DATI_ActualPosition"
   IOField "Campo I/O_3" at 227,176 size 96x30; FormatPattern 99999
      ProcessValue <- "IAI_DATI_Speed"
      Appearance <- "IAI_DATI_ErrSpeed"
   IOField "Campo I/O_4" at 227,105 size 96x30; FormatPattern s99999.999
      ProcessValue <- "Rugosimetro_Ra"
   IOField "Campo I/O_5" at 360,176 size 96x30; FormatPattern ??????????
      ProcessValue <- "SQL_SetName"
   Button "Pulsante_2" at 360,105 size 96x30; TextOff 'Simulation'; TextList "Read_Prof"
      on Release: ResetBit("Keyence_DATI_Activate")
      on Press: SetBit("Keyence_DATI_Activate")
      ProcessValue <- "Keyence_DATI_Request"
      Appearance <- "Keyence_DATI_Request"

screen "Segnalazioni" 480x272, template "Modello_1"
   AlarmView "Vista segnalazioni_1" at 3,47 size 474x196; AlarmLog "ErroriSql"

screen "SQL Report" 480x272, template "Modello_1"
   TextField "Casella di testo_2" at 8,52 size 202x20; Text 'Ciclo d'invio e acquisizione'
   IOField "Campo I/O_2" at 248,75 size 179x32; FormatPattern 99999
      ProcessValue <- "SQL_SendValue"
   TextField "Casella di testo_1" at 14,81 size 252x20; Text 'Tempo espresso in ms. 1000 = 1s'
   TextField "Casella di testo_3" at 8,114 size 138x20; Text 'Test connessione'
   TextField "Casella di testo_4" at 14,143 size 246x20; Text 'Determina lo stato del Database'
   TextField "Casella di testo_5" at 315,143 size 50x20; Text 'Online'
      Visibility <- "SQL_CheckState"
   TextField "Casella di testo_6" at 315,143 size 53x20; Text 'Offline'
      Visibility <- "SQL_CheckState"
   TextField "Casella di testo_7" at 8,176 size 91x20; Text 'Simulazione'
   IOField "Campo I/O_1" at 248,199 size 60x32; FormatPattern 999; Unit  A
      ProcessValue <- "Simulation_HighMax"
   TextField "Casella di testo_8" at 14,205 size 199x20; Text 'Imposta i parametri A-P-T'
   IOField "Campo I/O_3" at 305,199 size 56x32; FormatPattern 999; Unit  P
      ProcessValue <- "Simulation_PositionMax"
   IOField "Campo I/O_4" at 357,199 size 70x32; FormatPattern 99999; Unit  T
      ProcessValue <- "Simulation_SimuTimeIn"

screen "Home" 480x272, template "Modello_1"
   Softkey "Softkey_F2" at 0,0 size 0x0
      on KeyDown: StopRuntime(0)
   Button "Pulsante_4" at 40,59 size 104x67; TextOff 'JOG'
      on Click: ActivateScreen("JOG", 0)
   Button "Pulsante_1" at 188,59 size 104x67; TextOff 'Rugosimetro'
      on Click: ActivateScreen("Rugosimetro", 0)
   Button "Pulsante_2" at 336,59 size 104x67; TextOff 'Profilometro'
      on Click: ActivateScreen("Profilometro", 0)
   Button "Pulsante_3" at 336,143 size 104x68; TextOff 'SQL Report'
      on Click: ActivateScreen("SQL Report", 0)
   Button "Pulsante_5" at 188,143 size 104x68; TextOff 'Segnalazioni'
      on Click: ActivateScreen("Segnalazioni", 0)
   Button "Pulsante_6" at 40,143 size 104x68; TextOff 'Impostazioni'
      on Click: ActivateScreen("Impostazioni", 0)

screen "JOG" 480x272, template "Modello_1"
   Softkey "Softkey_F1" at 0,0 size 0x0
      on KeyUp: ResetBit("M_JOG_NEG")
      on KeyDown: SetBit("M_JOG_NEG")
   Softkey "Softkey_F2" at 0,0 size 0x0
      on KeyUp: ResetBit("M_RESET_ALLARM")
      on KeyDown: SetBit("M_RESET_ALLARM")
   Softkey "Softkey_F3" at 0,0 size 0x0
      on KeyUp: ResetBit("IL_100_ST")
      on KeyDown: SetBit("IL_100_ST")
   Softkey "Softkey_F4" at 0,0 size 0x0
      on KeyUp: ResetBit("M_JOG_POS")
      on KeyDown: SetBit("M_JOG_POS")
   IOField "Campo I/O_1" at 167,51 size 310x30; FormatPattern s999.99
      ProcessValue <- "IAI_DATI_ActualPosition"
   TextField "Casella di testo_1" at 6,56 size 162x20; Text 'Posizione attuale mm'
   IOField "Campo I/O_3" at 167,120 size 310x30; FormatPattern 99999
      ProcessValue <- "IAI_DATI_Speed_JOG"
   TextField "Casella di testo_3" at 6,125 size 145x20; Text 'Velocità in jog m/s'
   IOField "Campo I/O_4" at 167,190 size 310x30; FormatPattern 99
      ProcessValue <- "IAI_DATI_Aceleration_JOG"
   TextField "Casella di testo_4" at 6,195 size 156x20; Text 'Acelerazione m/s^2'
   IOField "Campo I/O_5" at 167,155 size 310x30; FormatPattern 99
      ProcessValue <- "IAI_DATI_Deceleration_JOG"
   TextField "Casella di testo_5" at 6,160 size 164x20; Text 'Decelerazione m/s^2'
   IOField "Campo I/O_2" at 167,85 size 310x30; FormatPattern s999.99
      ProcessValue <- "Keyence_DATI_MeasureValue"
   TextField "Casella di testo_2" at 6,90 size 139x20; Text 'Misura attuale um'

Template "Modello_1" 480x272
   GraphicView "Vista grafica_1" at 0,0 size 128x46; Picture "logo"
   TextField "Modello_Casella di testo_1" at 254,3 size 197x18; Text 'Banco prova - Profilometro'
   Circle "Modello_Cerchio_1" at 445,9 size 10x10
      Appearance <- "SQL_ChangeValue"
   Button "Modello_Pulsante_1" at 198,4 size 32x18; TextOff 'Text'; TextList "Jog/Auto"
      on Release: ResetBit("SelectOPMode")
      on Press: SetBit("SelectOPMode")
      ProcessValue <- "IAI_DATI_ModoOperativo"
   TextField "Modello_Casella di testo_5" at 131,3 size 67x18; Text 'OP Mode'
   AlarmView "Vista segnalazioni_1" at 129,23 size 348x20; AlarmLog "ErroriSql"
   Rectangle "Rettangolo_2" at 380,243 size 62x29
      Appearance <- "M_JOG_POS"
   Rectangle "Rettangolo_3" at 266,243 size 62x29
      Appearance <- "M_RESET_ALLARM"
   Rectangle "Rettangolo_5" at 38,243 size 62x29
      Appearance <- "M_JOG_NEG"
   TextField "Modello_Casella di testo_2" at 51,247 size 38x20; Text 'JOG-'
   TextField "Modello_Casella di testo_3" at 392,247 size 43x20; Text 'JOG+'
   GraphicView "Modello_Vista grafica_1" at 170,247 size 26x22; Picture "Grafica_1"
   TextField "Modello_Casella di testo_4" at 273,247 size 48x20; Text 'Reset'

screen "Impostazioni" 480x272, template "Modello_1"
   TextField "Casella di testo_3" at 60,130 size 65x20; Text 'Velocità'
   IOField "Campo I/O_5" at 197,154 size 96x32; FormatPattern 99
      ProcessValue <- "IAI_DATI_Deceleration"
      Appearance <- "IAI_DATI_ErrDeceleration"
   TextField "Casella di testo_5" at 194,130 size 109x20; Text 'Decelerazione'
   IOField "Campo I/O_8" at 329,154 size 96x32; FormatPattern s999999
      ProcessValue <- "IAI_DATI_ZonNeg"
      Appearance <- "IAI_DATI_ErrZoneNeg"
   TextField "Casella di testo_8" at 326,130 size 52x20; Text 'Zone -'
   TextField "Casella di testo_7" at 325,62 size 57x20; Text 'Zone +'
   IOField "Campo I/O_7" at 329,85 size 96x32; FormatPattern s999999
      ProcessValue <- "IAI_DATI_ZonePos"
      Appearance <- "IAI_DATI_ErrZonePos"
   IOField "Campo I/O_4" at 196,85 size 96x32; FormatPattern 99
      ProcessValue <- "IAI_DATI_Aceleration"
      Appearance <- "IAI_DATI_ErrAceleration"
   TextField "Casella di testo_4" at 195,62 size 101x20; Text 'Acelerazione'
   TextField "Casella di testo_2" at 60,62 size 105x20; Text 'Position Band'
   IOField "Campo I/O_2" at 61,85 size 96x32; FormatPattern 99999
      ProcessValue <- "IAI_DATI_PositionBand"
      Appearance <- "IAI_DATI_ErrPositionBand"
   IOField "Campo I/O_1" at 61,154 size 96x32; FormatPattern 99999
      ProcessValue <- "IAI_DATI_Speed"
      Appearance <- "IAI_DATI_ErrSpeed"

screen "Profilometro" 480x272, template "Modello_1"
   FunctionTrendControl "Vista delle curve f(x)_1" at 3,46 size 377x197
   Circle "Modello_Cerchio_1" at 454,125 size 10x10
      Appearance <- "Keyence_DATI_IsValid"
   TextField "Casella di testo_3" at 391,122 size 74x15; Text 'Rich. valida'
   TextField "Casella di testo_5" at 391,134 size 56x15; Text 'P.Errore'
   Circle "Modello_Cerchio_3" at 454,137 size 10x10
      Appearance <- "Keyence_DATI_IsError"
   IOField "Campo I/O_1" at 383,218 size 94x24; FormatPattern ??????????
      ProcessValue <- "SQL_SetName"
   TextField "Casella di testo_6" at 401,200 size 67x17; Text 'Nome Set'
   TextField "Casella di testo_7" at 391,162 size 88x17; Text 'Sql Send File'
   TextField "Casella di testo_4" at 391,146 size 63x15; Text 'Stato SQL'
   Circle "Modello_Cerchio_2" at 454,149 size 10x10
      Appearance <- "SQL_CheckState"
   IOField "Campo I/O_3" at 427,65 size 45x18; FormatPattern s99999.99
      ProcessValue <- "SQL_CTUAlt"
   IOField "Campo I/O_4" at 427,101 size 45x18; FormatPattern s99999.99
      ProcessValue <- "SQL_CTUPos"
   TextField "Casella di testo_9" at 439,49 size 24x17; Text 'Alt'
   TextField "Casella di testo_10" at 436,85 size 28x17; Text 'Pos'
   Button "Pulsante_4" at 386,65 size 37x18; TextOff 'Start'
      on Release: ResetBit("M_DSTR_ON")
      on Press: SetBit("M_DSTR_ON")
   IOField "Campo I/O_2" at 386,101 size 37x18; FormatPattern 99999
      ProcessValue <- "IAI_DATI_Speed"
      Appearance <- "IAI_DATI_ErrSpeed"
   TextField "Casella di testo_1" at 393,86 size 25x17; Text 'Vel'
   Button "Pulsante_3" at 398,181 size 65x16; TextOff 'Simulation'; TextList "SQLState"
      on Press: SetBit("SQL_BtnSend")
      on Release: ResetBit("SQL_BtnSend")
      ProcessValue <- "SQL_CheckState"

VB script "Report"
   ' -----------------------------------------------------------------------------------------------;
   ' Autore: Valentino Fabbri
   ' Data creazione: 16/09/2018
   ' Revisione: 1.5.0-30092018
   ' -----------------------------------------------------------------------------------------------;
   ' Inizio dichiarazioni --------------------------------------------------------------------------;
     Dim objConnection, str1, str2, strSQL2
     Dim objCommand, objRecordSet, strSQL0, strDirectory, strFile
     Dim NomeSet, Posizione, Misura, NomeFile, SQLState, fso, fo, MyFile, TextStreamTest
     Const ForReading = 1, ForWriting = 2
     Const conAdOpenStatic = 3 
     Const conAdLockOptimistic = 3
   ' Fine variabili --------------------------------------------------------------------------------;
   ' -----------------------------------------------------------------------------------------------;
   ' Query SQL -------------------------------------------------------------------------------------;
   
     'Valori RT
     'NomeSet = SmartTags("SQL_SetName")
     'Posizione = SmartTags("IAI_DATI_ActualPosition")
     'Misura = SmartTags("Keyence_DATI_PresentValue")
     Set fso = CreateObject("FileCtl.FileSystem")
     Set fo = CreateObject("FileCtl.File")
     
     Set NomeFile = SmartTags("SQL_SetName")
     
     strDirectory = "\MeasureData\" + NomeFile + ".sql"
             	 
     On Error Resume Next 'Catturo gli errori ed eseguo la riga successiva
   
     Set objConnection = CreateObject("ADOCE.Connection")
     Set objRecordSet = CreateObject("ADOCE.RecordSet")
     'Set objCommand = CreateObject("ADOCE.Command")
     
     objConnection.ConnectionString = "DRIVER=\windows\dbodbc10.dll; UID=sa; PWD=fiesta92; Integrated=No;" &_
   								 "AutoStop=Yes; EngineName=Artec; LINKS=tcpip(host=18.100.70.1;port=2638;" &_
   								 "dobroadcast=none; LOG=\sa_connection.txt; START=dbsrv10 -c 8M)" 
   								 
     objConnection.Open 'Apro la connessione
     Set MyFile = fo.Open(strDirectory, 1, ForReading)
     'TextStreamTest = MyFile.ReadAll
     
     If Err.Number <> 0 Then 'Vengono intercettati tutti gli errori SQL
     	bfde4b54-0db7-4817-8032-87127bf19bb9 "SQL Connection Error N#" & Err.Number & " - " & Err.Description
   	Err.Clear
   	'ServerOffline DB, TB 'Se c'è mancata connessione salvo i dati offline
   	Exit Sub
     End If
     
     If objConnection.State = 1 Then
     	objRecordSet.Open MyFile , objConnection, conAdOpenStatic, conAdLockOptimistic
       bfde4b54-0db7-4817-8032-87127bf19bb9 "Il comando SQL " & NomeFile & " è stato eseguito."
     End If
   
     If Err.Number <> 0 Then
     	bfde4b54-0db7-4817-8032-87127bf19bb9 "SQL Command Error N#" & Err.Number & " - " & Err.Description
   	Err.Clear 
   	Exit Sub
     End If 
     
     Set objConnection = Nothing 
     Set objRecordSet = Nothing
     'Set objCommand = Nothing
   ' Fine Query SQL --------------------------------------------------------------------------------;

VB script "ReportOffline"
   ' -----------------------------------------------------------------------------------------------;
   ' Autore: Valentino Fabbri
   ' Data creazione: 28/09/2018
   ' Revisione: 2.0.11-24102018
   ' Nota: 
   ' -----------------------------------------------------------------------------------------------;
   ' Inizio variabili ------------------------------------------------------------------------------;
     Dim NomeSet, Posizione, Misura
     Dim objFSO, objFO
     Dim strDirectory, strFile, strText
     Dim strTime
     Const ForAppending = 8
   ' Fine variabili --------------------------------------------------------------------------------;
   ' -----------------------------------------------------------------------------------------------;
   ' Inizio tempo in ms ----------------------------------------------------------------------------;
     strTime = NowMs() '& ""
   ' Fine tempo in ms ------------------------------------------------------------------------------;
   ' -----------------------------------------------------------------------------------------------;
   ' Inizio script ---------------------------------------------------------------------------------;
     'Valori RT
     NomeSet = SmartTags("SQL_SetName")
     Posizione = SmartTags("IAI_DATI_ActualPosition")
     Misura = SmartTags("Keyence_DATI_MeasureValue")
   
     'strDirectory = "\Storage Card USB\MeasureData" sulla chiavetta
     strDirectory = "\\PORT-54\Users\r.walia\Documents\Profilometro\Misure" ' sulla rete
     strFile = "\" & NomeSet & ".sql"
     strText = "INSERT INTO Profilometro (Posizione, Misura, NomeSet, Date)" 
     strText = strText	& " VALUES ( " & Posizione & "," & Misura & "," & "'" & NomeSet & "'," & "'" & strTime & "'" & ")"
   
     'Creo l'oggetto
     Set objFSO = CreateObject("FileCtl.FileSystem")
     Set objFO = CreateObject("FileCtl.File")
     
     If Err.Number <> 0 Then
   	  bfde4b54-0db7-4817-8032-87127bf19bb9 "Errore in R:23-34 " & CStr(Err.Number) & " " & Err.Description
   	  Err.Clear
   	  Exit Sub
     End If   
     
     On Error Resume Next
      
     If objFSO.Dir (strDirectory)<>"" Then
   	 ' la cartella MeasureData esiste
        If objFSO.Dir (strDirectory & strFile)<>"" Then
              objFO.Open strDirectory & strFile,8
              If Err.Number <> 0 Then
   	  	      bfde4b54-0db7-4817-8032-87127bf19bb9 "Errore in R:47 - N# " & CStr(Err.Number) & " " & Err.Description
   	          Err.Clear
   	          Exit Sub
              End If
        End If
     Else
      ' creo la cartella se non esiste
        objFSO.MkDir (strDirectory)
        ' apro il file
        objFO.Open strDirectory & strFile,8
        If Err.Number <> 0 Then
   	    bfde4b54-0db7-4817-8032-87127bf19bb9 "Errore in R:58 - N# " & CStr(Err.Number) & " " & Err.Description
   	    Err.Clear
   	    Exit Sub
        End If
     End If
     
     If objFO.LOF = 0 Then
   	 objFO.LinePrint(strText)
   	 If Err.Number <> 0 Then
   	    bfde4b54-0db7-4817-8032-87127bf19bb9 "Errore in R:67 - N# " & CStr(Err.Number) & " " & Err.Description
   	    Err.Clear
   	    Exit Sub
        End If
     Else
   	 objFO.LinePrint(strText)
   	 If Err.Number <> 0 Then
   	    bfde4b54-0db7-4817-8032-87127bf19bb9 "Errore in R:74 - N# " & CStr(Err.Number) & " " & Err.Description
   	    Err.Clear
   	    Exit Sub
        End If
     End If
     
     Set objFSO = Nothing
     Set objFO = Nothing
     

VB script "NowMs"
   ' Inizio variabili --------------------------------------------------------------------------------;
    Dim t, temp, Miliseconds, Seconds, Minutes, Hours, strTime, dd, mm, yy, n
   ' Fine variabili ----------------------------------------------------------------------------------;
   ' -------------------------------------------------------------------------------------------------;
   ' Inizio tempo in ms ------------------------------------------------------------------------------;
     dd = Digits(Day(Date()),2)
     mm = Digits(Month(Date()),2)
     yy = Digits(Right(Year(Date()),2),2)
     t = Timer
     temp = Int(t)
   
     Miliseconds = Int((t-temp) * 1000)
     
     Seconds = temp Mod 60
     temp    = Int(temp/60)
     Minutes = temp Mod 60
     Hours   = Int(temp/60)
   ' Formato
     strTime =           String(2 - Len(dd), "0") & dd & "-"
     strTime = strTime & String(2 - Len(mm), "0") & mm & "-"
     strTime = strTime & String(2 - Len(yy), "0") & yy & " "
     strTime = strTime & String(2 - Len(Hours), "0") & Hours & ":"
     strTime = strTime & String(2 - Len(Minutes), "0") & Minutes & ":"
     strTime = strTime & String(2 - Len(Seconds), "0") & Seconds & "."
     strTime = strTime & String(4 - Len(Miliseconds), "0") & Miliseconds
     NowMs = strTime
   ' Fine tempo in ms --------------------------------------------------------------------------------;
   ' -------------------------------------------------------------------------------------------------;

VB script "Digits"
   If totalDigits > Len(n) Then 
   	Digits = String(totalDigits-Len(n),"0") & n 
   Else 
       Digits = n 
   End If 

VB script "CheckState"
   Dim objConnection, myConnection
   
   On Error Resume Next 'Catturo gli errori ed eseguo la riga successiva
   
   Set objConnection = CreateObject("ADODB.Connection")
   
   myConnection = "Provider=MSDASQL; DSN=Artec; UID=sa; PWD=fiesta92; Initial Catalog=Artec"
   
   objConnection.ConnectionString = myConnection
   objConnection.Open 'Apro la connessione
      
   If Err.Number <> 0 Then 'Vengono intercettati tutti gli errori SQL
     bfde4b54-0db7-4817-8032-87127bf19bb9 "SQL Connection Error N#" & Err.Number & " - " & Err.Description
     Err.Clear
     Exit Sub
   End If
     
   If objConnection.State = 1 Then 
     SmartTags("SQL_CheckState") = 1
   Else
     SmartTags("SQL_CheckState") = 0	  
   End If	
   
   If Err.Number <> 0 Then
     bfde4b54-0db7-4817-8032-87127bf19bb9 "SQL Command Error N#" & Err.Number & " - " & Err.Description
     Err.Clear 
     Exit Sub
   End If 
   Set objConnection = Nothing 

VB script "DataLogPc"
   ' -----------------------------------------------------------------------------------------------;
   ' Autore: Valentino Fabbri
   ' Data creazione: 29/09/2018
   ' Revisione: 2.0.00-29092018
   ' Nota: Da ora è possibile in caso di mancata connessione salvare i dati offline ed inserirli dopo nel db
   ' -----------------------------------------------------------------------------------------------;
   ' Inizio variabili ------------------------------------------------------------------------------;
     Dim strSQL2
     Dim NomeSet, Posizione, Misura
     Dim objFSO, objFolder, objShell, objTextFile, objFile
     Dim strDirectory, strFile, strText
     Dim t, temp, Miliseconds, Seconds, Minutes, Hours, strTime
   ' Fine variabili --------------------------------------------------------------------------------;
   ' -----------------------------------------------------------------------------------------------;
   ' Inizio tempo in ms --------------------------------------------------------------------------------;
     strTime = NowMs() '& ""
   ' Fine tempo in ms --------------------------------------------------------------------------------;
   ' -----------------------------------------------------------------------------------------------;
   ' Inizio script --------------------------------------------------------------------------------;
     'Valori RT
     NomeSet = SmartTags("SQL_SetName")
     Posizione = SmartTags("IAI_DATI_ActualPosition")
     Misura = SmartTags("Keyence_DATI_MeasureValue")
     
     'Option Explicit
     strDirectory = "C:\Storage Card SD\MeasureData"
     strFile = "\" & NomeSet & ".sql"
     strText = "INSERT INTO Profilometro (Posizione, Misura, NomeSet, Date)" & _
               "VALUES ( " & "'" & Posizione & "'," & "'" & Misura & "'," & "'" & NomeSet & "'," & "'" & strTime & "'" & ")"
   
     'Creo l'oggetto
     Set objFSO = CreateObject("Scripting.FileSystemObject")
     On Error Resume Next
     'La cartella esiste?
     If objFSO.FolderExists(strDirectory) Then
        Set objFolder = objFSO.GetFolder(strDirectory)     
     'La creo
     Else
        Set objFolder = objFSO.CreateFolder(strDirectory)
     End If
     
     'Il file esiste?
     If objFSO.FileExists(strDirectory & strFile) Then
        Set objFolder = objFSO.GetFolder(strDirectory)
     'Lo creo
     Else
        Set objFile = objFSO.CreateTextFile(strDirectory & strFile)
     End If
   
     Set objFile = Nothing
     Set objFolder = Nothing
     
     'ForAppending = 8 ForReading = 1, ForWriting = 2
     Const ForAppending = 8
   
     Set objTextFile = objFSO.OpenTextFile _
     (strDirectory & strFile, ForAppending, True)
   
     'Scrivo strText ogni volta che eseguo lo script
     objTextFile.WriteLine(strText)
     If Err.Number <> 0 Then
     	bfde4b54-0db7-4817-8032-87127bf19bb9 "Write Error - R:63 - N#" & Err.Number & " - " & Err.Description
   	Err.Clear 
   	Exit Sub
     End If 
     
     objTextFile.Close

VB script "DataLogOnline"
   ' -----------------------------------------------------------------------------------------------;
   ' Autore: Valentino Fabbri
   ' Data creazione: 16/09/2018
   ' Revisione: 1.6.0-23102018
   ' -----------------------------------------------------------------------------------------------;
   ' Inizio dichiarazioni --------------------------------------------------------------------------;
     Dim objConnection, connString, str1, str2, strSQL2
     Dim objCommand, objRecordSet, strSQL0, strDirectory, strFile
     Dim NomeSet, Posizione, Misura, NomeFile, SQLState, fso, MyFile, TextStreamTest
     Const ForReading = 1, ForWriting = 2
     Const conAdOpenStatic = 3 
     Const conAdLockOptimistic = 3
   ' Fine variabili --------------------------------------------------------------------------------;
   ' -----------------------------------------------------------------------------------------------;
   ' Query SQL -------------------------------------------------------------------------------------;
     Set fso = CreateObject("Scripting.FileSystemObject")
     NomeFile = SmartTags("SQL_SetName")
     connString = "Provider=MSDASQL; DSN=Artec; UID=sa; PWD=fiesta92; Initial Catalog=Artec"
     strDirectory = "C:\Storage Card SD\MeasureData\" + NomeFile + ".sql"
                   	 
     On Error Resume Next 'Catturo gli errori ed eseguo la riga successiva
   
     Set objConnection = CreateObject("ADODB.Connection")
     Set objRecordSet = CreateObject("ADODB.Recordset")
     Set objCommand = CreateObject("ADODB.Command")
     
     'Il file esiste?
     If fso.FileExists(strDirectory & strFile) Then
        Set MyFile = fso.OpenTextFile(strDirectory, ForReading)
        TextStreamTest = MyFile.ReadAll
        objConnection.CommandTimeout = 900
        objConnection.ConnectionString = connString
        objConnection.Open 'Apro la connessione
        If objConnection.State = 1 Then
     	    objRecordSet.Open TextStreamTest , objConnection, conAdOpenStatic, conAdLockOptimistic
           bfde4b54-0db7-4817-8032-87127bf19bb9 "Il comando SQL " & NomeFile & " è stato eseguito."
           If Err.Number <> 0 Then 'Vengono intercettati tutti gli errori SQL
     	       bfde4b54-0db7-4817-8032-87127bf19bb9 "SQL Connection Error - R:36 - N#" & Err.Number & " - " & Err.Description
   	       Err.Clear
   	       Exit Sub
           End If
   	 Else
   		 bfde4b54-0db7-4817-8032-87127bf19bb9 "SQL Connection Error - R:34 - N#" & Err.Number & " - " & "Il Server non è disponibile"
   		 Err.Clear
   		 Exit Sub
        End If
     Else
        bfde4b54-0db7-4817-8032-87127bf19bb9 "Read Error - R:21 - N#404 - La query non è presente"
   	 Err.Clear
   	 Exit Sub
     End If
     
     If Err.Number <> 0 Then 'Vengono intercettati tutti gli errori SQL
     	bfde4b54-0db7-4817-8032-87127bf19bb9 "Unhandled Error - R:53 - N#" & Err.Number & " - " & Err.Description
   	Err.Clear
   	Exit Sub
     End If
     
     Set objConnection = Nothing 
     Set objRecordSet = Nothing
     Set objCommand = Nothing
   ' Fine Query SQL --------------------------------------------------------------------------------;

VB script "CheckCollision"
   If SmartTags("Keyence_DATI_ReadError") = 1 Then
   	bfde4b54-0db7-4817-8032-87127bf19bb9("Collisione fallita.")
   Else
   	bfde4b54-0db7-4817-8032-87127bf19bb9("Misura iniziata.")
   End If

VB script "ShowError"
   Dim Compare
   Compare = SmartTags(Parametro)
   If (Compare > ValoreAlto Or Compare < ValoreBasso) Then
   	SmartTags(Errore) = 1
   Else
   	SmartTags(Errore) = 0
   End If

VB script "ReportOffline_backup"
   ' -----------------------------------------------------------------------------------------------;
   ' Autore: Valentino Fabbri
   ' Data creazione: 28/09/2018
   ' Revisione: 2.0.11-24102018
   ' Nota: 
   ' -----------------------------------------------------------------------------------------------;
   ' Inizio variabili ------------------------------------------------------------------------------;
     Dim NomeSet, Posizione, Misura
     Dim objFSO, objFO
     Dim strDirectory, strFile, strText
     Dim strTime
     Const ForAppending = 8
   ' Fine variabili --------------------------------------------------------------------------------;
   ' -----------------------------------------------------------------------------------------------;
   ' Inizio tempo in ms ----------------------------------------------------------------------------;
     strTime = NowMs() '& ""
   ' Fine tempo in ms ------------------------------------------------------------------------------;
   ' -----------------------------------------------------------------------------------------------;
   ' Inizio script ---------------------------------------------------------------------------------;
     'Valori RT
     NomeSet = SmartTags("SQL_SetName")
     Posizione = SmartTags("IAI_DATI_ActualPosition")
     Misura = SmartTags("Keyence_DATI_MeasureValue")
   
     'strDirectory = "\Storage Card USB\MeasureData" sulla chiavetta
     strDirectory = "\\PORT-54\Users\r.walia\Documents\Profilometro\Misure" ' sulla rete
     strFile = "\" & NomeSet & ".sql"
     strText = "INSERT INTO Profilometro (Posizione, Misura, NomeSet, Date)" 
     strText = strText	& " VALUES ( " & "'" & Posizione & "'," & "'" & Misura & "'," & "'" & NomeSet & "'," & "'" & strTime & "'" & ")"
   
     'Creo l'oggetto
     Set objFSO = CreateObject("FileCtl.FileSystem")
     Set objFO = CreateObject("FileCtl.File")
     
     If Err.Number <> 0 Then
   	  bfde4b54-0db7-4817-8032-87127bf19bb9 "Errore in R:23-34 " & CStr(Err.Number) & " " & Err.Description
   	  Err.Clear
   	  Exit Sub
     End If   
     
     On Error Resume Next
      
     If objFSO.Dir (strDirectory)<>"" Then
   	 ' la cartella MeasureData esiste
        If objFSO.Dir (strDirectory & strFile)<>"" Then
              objFO.Open strDirectory & strFile,8
              If Err.Number <> 0 Then
   	  	      bfde4b54-0db7-4817-8032-87127bf19bb9 "Errore in R:47 - N# " & CStr(Err.Number) & " " & Err.Description
   	          Err.Clear
   	          Exit Sub
              End If
        End If
     Else
      ' creo la cartella se non esiste
        objFSO.MkDir (strDirectory)
        ' apro il file
        objFO.Open strDirectory & strFile,8
        If Err.Number <> 0 Then
   	    bfde4b54-0db7-4817-8032-87127bf19bb9 "Errore in R:58 - N# " & CStr(Err.Number) & " " & Err.Description
   	    Err.Clear
   	    Exit Sub
        End If
     End If
     
     If objFO.LOF = 0 Then
   	 objFO.LinePrint(strText)
   	 If Err.Number <> 0 Then
   	    bfde4b54-0db7-4817-8032-87127bf19bb9 "Errore in R:67 - N# " & CStr(Err.Number) & " " & Err.Description
   	    Err.Clear
   	    Exit Sub
        End If
     Else
   	 objFO.LinePrint(strText)
   	 If Err.Number <> 0 Then
   	    bfde4b54-0db7-4817-8032-87127bf19bb9 "Errore in R:74 - N# " & CStr(Err.Number) & " " & Err.Description
   	    Err.Clear
   	    Exit Sub
        End If
     End If
     
     Set objFSO = Nothing
     Set objFO = Nothing
     

scheduled task "Check SQL State"
   on Action: "CheckState"()
   Triggers <- "1 min"
*)